C03640=1043.062,430.880,361.254,175.358,44.997,159.099
C03641=1043.073,431.124,361.204,175.371,45.006,159.102
C03642=1043.084,431.369,361.154,175.384,45.014,159.106
C03643=1043.096,431.614,361.104,175.397,45.023,159.110
C03644=1043.107,431.859,361.054,175.411,45.031,159.113
C03645=1043.119,432.104,361.004,175.424,45.040,159.117
C03646=1043.130,432.348,360.954,175.437,45.048,159.121
C03647=1043.142,432.593,360.904,175.450,45.057,159.125
C03648=1043.153,432.837,360.853,175.463,45.065,159.128
C03649=1043.165,433.082,360.803,175.477,45.074,159.132
C03650=1043.177,433.326,360.752,175.491,45.083,159.136
C03651=1043.188,433.571,360.701,175.504,45.092,159.140
C03652=1043.200,433.815,360.652,175.517,45.100,159.144
C03653=1043.212,434.060,360.601,175.531,45.109,159.147
C03654=1043.223,434.288,360.554,175.543,45.117,159.151
C03655=1043.234,434.517,360.506,175.556,45.125,159.155
C03656=1043.245,434.745,360.459,175.570,45.133,159.158
C03657=1043.256,434.972,360.411,175.581,45.142,159.162
C03658=1043.267,435.201,360.364,175.595,45.150,159.166
C03659=1043.278,435.429,360.317,175.608,45.158,159.169
C03660=1043.290,435.657,360.269,175.621,45.166,159.173
C03661=1043.301,435.885,360.222,175.634,45.175,159.177
C03662=1043.312,436.130,360.171,175.647,45.184,159.181
C03663=1043.324,436.374,360.119,175.662,45.193,159.185
C03664=1043.335,436.618,360.068,175.675,45.202,159.189
C03665=1043.348,436.862,360.018,175.690,45.211,159.193
C03666=1043.360,437.107,359.966,175.704,45.220,159.197
C03667=1043.372,437.351,359.915,175.718,45.229,159.201
C03668=1043.384,437.597,359.863,175.732,45.238,159.205
C03669=1043.397,437.840,359.811,175.747,45.247,159.209
C03670=1043.408,438.085,359.759,175.761,45.257,159.213
C03671=1043.420,438.329,359.708,175.775,45.266,159.217
C03672=1043.432,438.573,359.656,175.790,45.275,159.222
C03673=1043.445,438.818,359.605,175.805,45.284,159.226
C03674=1043.457,439.061,359.553,175.820,45.294,159.230
C03675=1043.469,439.306,359.502,175.835,45.303,159.234
C03676=1043.481,439.550,359.449,175.848,45.313,159.238
C03677=1043.494,439.794,359.397,175.863,45.322,159.243
C03678=1043.506,440.039,359.346,175.878,45.332,159.247
C03679=1043.518,440.283,359.293,175.893,45.341,159.251
C03680=1043.531,440.527,359.241,175.908,45.350,159.256
C03681=1043.543,440.771,359.189,175.923,45.360,159.260
C03682=1043.555,441.015,359.137,175.938,45.370,159.264
C03683=1043.568,441.260,359.084,175.953,45.379,159.269
C03684=1043.580,441.504,359.032,175.969,45.389,159.273
C03685=1043.593,441.748,358.980,175.984,45.399,159.277
C03686=1043.605,441.992,358.928,176.000,45.408,159.282
C03687=1043.618,442.236,358.874,176.015,45.418,159.286
C03688=1043.631,442.480,358.822,176.030,45.428,159.291
C03689=1043.643,442.725,358.770,176.045,45.437,159.295
C03690=1043.655,442.968,358.716,176.062,45.447,159.300
C03691=1043.668,443.213,358.664,176.077,45.457,159.304
C03692=1043.681,443.457,358.611,176.092,45.467,159.309
C03693=1043.694,443.700,358.558,176.109,45.476,159.313
C03694=1043.706,443.945,358.505,176.124,45.486,159.318
C03695=1043.719,444.189,358.452,176.140,45.496,159.322
C03696=1043.732,444.433,358.399,176.156,45.506,159.327
C03697=1043.746,444.677,358.346,176.171,45.516,159.332
C03698=1043.758,444.920,358.293,176.188,45.527,159.337
C03699=1043.772,445.162,358.240,176.205,45.536,159.341
C03700=1043.784,445.405,358.187,176.220,45.546,159.346
C03701=1043.799,445.650,358.135,176.237,45.556,159.350
C03702=1043.813,445.893,358.084,176.253,45.566,159.355
C03703=1043.828,446.136,358.032,176.269,45.575,159.360
C03704=1043.845,446.380,357.982,176.286,45.585,159.364
C03705=1043.861,446.624,357.931,176.302,45.594,159.369
C03706=1043.879,446.867,357.882,176.319,45.603,159.373
C03707=1043.896,447.112,357.833,176.336,45.613,159.378
C03708=1043.915,447.355,357.784,176.353,45.621,159.382
C03709=1043.934,447.601,357.735,176.369,45.630,159.387
C03710=1043.954,447.845,357.687,176.386,45.639,159.391
C03711=1043.974,448.089,357.641,176.403,45.648,159.396
C03712=1043.995,448.334,357.593,176.420,45.656,159.400
C03713=1044.016,448.578,357.547,176.438,45.665,159.404
C03714=1044.054,448.991,357.470,176.467,45.678,159.412
C03715=1044.094,449.404,357.395,176.496,45.692,159.419
C03716=1044.135,449.817,357.321,176.526,45.706,159.426
C03717=1044.178,450.231,357.248,176.556,45.718,159.433
C03718=1044.204,450.476,357.205,176.574,45.726,159.438
C03719=1044.231,450.722,357.163,176.591,45.733,159.442
C03720=1044.259,450.968,357.122,176.610,45.741,159.446
C03721=1044.287,451.213,357.081,176.627,45.748,159.450
C03722=1043.984,451.252,356.769,176.629,45.829,159.475
C03723=1043.956,451.007,356.810,176.612,45.822,159.470
C03724=1043.927,450.761,356.851,176.593,45.815,159.466
C03725=1043.901,450.516,356.893,176.575,45.808,159.462
C03726=1043.874,450.271,356.936,176.558,45.800,159.458
C03727=1043.833,449.874,357.005,176.528,45.788,159.451
C03728=1043.793,449.476,357.076,176.500,45.775,159.444
C03729=1043.754,449.080,357.149,176.471,45.763,159.437
C03730=1043.717,448.682,357.223,176.443,45.749,159.430
C03731=1043.695,448.438,357.268,176.426,45.741,159.426
C03732=1043.674,448.193,357.315,176.408,45.733,159.421
C03733=1043.654,447.949,357.362,176.391,45.724,159.417
C03734=1043.633,447.704,357.410,176.374,45.716,159.412
C03735=1043.614,447.460,357.458,176.358,45.706,159.408
C03736=1043.595,447.216,357.506,176.341,45.698,159.403
C03737=1043.577,446.972,357.554,176.324,45.689,159.399
C03738=1043.559,446.727,357.605,176.307,45.680,159.394
C03739=1043.542,446.484,357.654,176.290,45.671,159.390
C03740=1043.526,446.240,357.705,176.274,45.662,159.385
C03741=1043.511,445.997,357.756,176.257,45.652,159.381
C03742=1043.496,445.753,357.807,176.241,45.643,159.376
C03743=1043.481,445.510,357.859,176.225,45.633,159.372
C03744=1043.467,445.266,357.912,176.208,45.623,159.367
C03745=1043.454,445.023,357.964,176.193,45.613,159.362
C03746=1043.441,444.781,358.017,176.176,45.603,159.358
C03747=1043.421,444.396,358.101,176.151,45.587,159.350
C03748=1043.400,444.010,358.184,176.125,45.572,159.343
C03749=1043.380,443.625,358.269,176.100,45.556,159.336
C03750=1043.360,443.240,358.352,176.075,45.541,159.329
C03751=1043.347,442.995,358.405,176.060,45.531,159.324
C03752=1043.334,442.752,358.457,176.044,45.522,159.320
C03753=1043.322,442.508,358.510,176.028,45.512,159.315
C03754=1043.309,442.264,358.563,176.013,45.502,159.310
C03755=1043.296,442.020,358.615,175.998,45.493,159.306
C03756=1043.284,441.776,358.667,175.982,45.483,159.302
C03757=1043.271,441.532,358.721,175.967,45.474,159.297
C03758=1043.259,441.288,358.773,175.952,45.464,159.293
C03759=1043.246,441.043,358.825,175.936,45.454,159.288
C03760=1043.234,440.800,358.877,175.921,45.445,159.284
C03761=1043.221,440.555,358.930,175.906,45.436,159.280
C03762=1043.209,440.311,358.982,175.891,45.426,159.275
C03763=1043.197,440.067,359.033,175.876,45.417,159.271
C03764=1043.184,439.822,359.086,175.861,45.407,159.267
C03765=1043.172,439.578,359.138,175.846,45.398,159.263
C03766=1043.160,439.334,359.190,175.832,45.389,159.258
C03767=1043.147,439.089,359.242,175.817,45.379,159.254
C03768=1043.135,438.845,359.294,175.802,45.370,159.250
C03769=1043.123,438.601,359.345,175.788,45.361,159.246
C03770=1043.111,438.357,359.397,175.773,45.351,159.241
C03771=1043.099,438.112,359.449,175.758,45.342,159.237
C03772=1043.087,437.868,359.500,175.744,45.334,159.233
C03773=1043.074,437.624,359.552,175.730,45.324,159.229
C03774=1043.062,437.380,359.603,175.715,45.315,159.225
C03775=1043.051,437.135,359.655,175.701,45.306,159.221
C03776=1043.039,436.891,359.706,175.687,45.297,159.217
C03777=1043.027,436.646,359.757,175.672,45.288,159.213
C03778=1043.014,436.402,359.808,175.659,45.279,159.209
C03779=1043.002,436.157,359.860,175.644,45.270,159.205
C03780=1042.990,435.913,359.911,175.631,45.261,159.201
C03781=1042.979,435.668,359.962,175.616,45.252,159.197
C03782=1042.967,435.423,360.013,175.603,45.243,159.193
C03783=1042.951,435.108,360.079,175.584,45.232,159.188
C03784=1042.936,434.791,360.145,175.567,45.221,159.183
C03785=1042.920,434.475,360.210,175.548,45.209,159.178
C03786=1042.905,434.158,360.276,175.531,45.198,159.173
C03787=1042.894,433.913,360.326,175.517,45.189,159.169
C03788=1042.881,433.669,360.377,175.504,45.181,159.165
C03789=1042.870,433.424,360.428,175.490,45.172,159.161
C03790=1042.858,433.180,360.477,175.476,45.164,159.157
C03791=1042.847,432.935,360.528,175.463,45.155,159.153
C03792=1042.835,432.691,360.578,175.450,45.147,159.150
C03793=1042.823,432.446,360.628,175.437,45.138,159.146
C03794=1042.812,432.201,360.679,175.424,45.130,159.142
C03795=1042.800,431.956,360.729,175.411,45.121,159.138
C03796=1042.789,431.712,360.779,175.396,45.113,159.135
C03797=1042.777,431.467,360.829,175.383,45.104,159.131
C03798=1042.766,431.223,360.880,175.370,45.096,159.127
C03799=1042.754,430.978,360.930,175.357,45.087,159.124
C03800=1042.743,430.733,360.979,175.345,45.079,159.120
C03801=1042.732,430.488,361.030,175.332,45.071,159.116
C03802=1042.720,430.244,361.079,175.319,45.062,159.113
C03803=1042.709,429.998,361.129,175.306,45.054,159.109
C03804=1042.697,429.754,361.179,175.293,45.046,159.105
C03805=1042.686,429.509,361.229,175.280,45.037,159.102
C03806=1042.675,429.265,361.279,175.267,45.029,159.098
C03807=1042.664,429.020,361.328,175.255,45.021,159.095
C03808=1042.653,428.774,361.378,175.243,45.013,159.091
C03809=1042.641,428.530,361.427,175.229,45.005,159.087
C03810=1042.630,428.285,361.477,175.217,44.997,159.084
C03811=1042.619,428.040,361.526,175.205,44.989,159.081
C03812=1042.608,427.796,361.575,175.192,44.981,159.077
C03813=1042.597,427.551,361.625,175.179,44.973,159.074
C03814=1042.586,427.306,361.674,175.168,44.964,159.070
C03815=1042.574,427.061,361.723,175.155,44.957,159.067
C03816=1042.563,426.816,361.771,175.142,44.949,159.063
C03817=1042.552,426.571,361.821,175.131,44.941,159.060
C03818=1042.541,426.326,361.870,175.118,44.933,159.056
C03819=1042.530,426.081,361.919,175.106,44.925,159.053
C03820=1042.519,425.836,361.968,175.094,44.917,159.050
C03821=1042.508,425.591,362.017,175.082,44.909,159.046
C03822=1042.497,425.347,362.065,175.070,44.902,159.043
C03823=1042.487,425.101,362.114,175.058,44.894,159.040
C03824=1042.475,424.856,362.163,175.045,44.886,159.036
C03825=1042.464,424.611,362.212,175.034,44.878,159.033
C03826=1042.454,424.366,362.260,175.022,44.870,159.030
C03827=1042.443,424.121,362.309,175.010,44.863,159.026
C03828=1042.432,423.876,362.358,174.998,44.855,159.023
C03829=1042.421,423.631,362.406,174.987,44.847,159.020
C03830=1042.410,423.386,362.454,174.974,44.840,159.017
C03831=1042.399,423.141,362.502,174.963,44.833,159.013
C03832=1042.388,422.895,362.550,174.952,44.825,159.010
C03833=1042.377,422.651,362.599,174.941,44.817,159.007
C03834=1042.366,422.405,362.647,174.928,44.810,159.004
C03835=1042.356,422.161,362.694,174.917,44.803,159.001
C03836=1042.345,421.915,362.743,174.905,44.795,158.997
C03837=1042.334,421.671,362.791,174.894,44.787,158.994
C03838=1042.323,421.425,362.839,174.883,44.780,158.991
C03839=1042.314,421.205,362.882,174.872,44.773,158.988
C03840=1042.304,420.985,362.925,174.862,44.767,158.986
C03841=1042.295,420.765,362.968,174.852,44.760,158.983
C03842=1042.286,420.546,363.011,174.842,44.754,158.980
C03843=1042.276,420.327,363.054,174.832,44.747,158.977
C03844=1042.267,420.106,363.097,174.822,44.740,158.974
C03845=1042.257,419.886,363.140,174.811,44.734,158.972
C03846=1042.248,419.666,363.182,174.802,44.728,158.969
C03847=1042.237,419.421,363.230,174.791,44.720,158.966
C03848=1042.227,419.176,363.278,174.779,44.713,158.963
C03849=1042.217,418.930,363.325,174.768,44.705,158.960
C03850=1042.206,418.686,363.373,174.757,44.699,158.957
C03851=1042.196,418.440,363.420,174.747,44.691,158.954
C03852=1042.186,418.195,363.467,174.736,44.684,158.951
C03853=1042.175,417.950,363.515,174.725,44.677,158.948
C03854=1042.165,417.704,363.562,174.714,44.670,158.945
C03855=1042.154,417.459,363.609,174.703,44.663,158.942
C03856=1042.144,417.213,363.656,174.692,44.656,158.939
C03857=1042.133,416.968,363.703,174.681,44.649,158.936
C03858=1042.123,416.723,363.751,174.671,44.642,158.933
C03859=1042.112,416.478,363.797,174.660,44.635,158.930
C03860=1042.102,416.233,363.844,174.649,44.628,158.927
C03861=1042.092,415.987,363.892,174.638,44.621,158.924
C03862=1042.081,415.741,363.938,174.628,44.614,158.922
C03863=1042.071,415.496,363.985,174.618,44.607,158.919
C03864=1042.061,415.251,364.032,174.607,44.601,158.916
C03865=1042.051,415.005,364.078,174.597,44.594,158.913
C03866=1042.041,414.760,364.126,174.586,44.587,158.910
C03867=1042.030,414.514,364.172,174.575,44.580,158.907
C03868=1042.020,414.269,364.219,174.565,44.573,158.905
C03869=1042.010,414.023,364.265,174.555,44.566,158.902
C03870=1042.000,413.778,364.312,174.545,44.559,158.899
C03871=1041.989,413.532,364.358,174.534,44.553,158.896
C03872=1041.980,413.288,364.405,174.525,44.546,158.893
C03873=1041.970,413.042,364.452,174.514,44.540,158.891
C03874=1041.960,412.796,364.498,174.504,44.532,158.888
C03875=1041.949,412.550,364.544,174.494,44.526,158.885
C03876=1041.940,412.306,364.591,174.484,44.520,158.883
C03877=1041.930,412.060,364.637,174.473,44.513,158.880
C03878=1041.919,411.814,364.683,174.463,44.506,158.877
C03879=1041.910,411.569,364.730,174.453,44.500,158.874
C03880=1041.899,411.323,364.775,174.443,44.493,158.872
C03881=1041.889,411.078,364.822,174.434,44.487,158.869
C03882=1041.880,410.832,364.867,174.423,44.480,158.866
C03883=1041.869,410.586,364.913,174.414,44.474,158.864
C03884=1041.859,410.341,364.959,174.403,44.467,158.861
C03885=1041.849,410.096,365.005,174.393,44.461,158.858
C03886=1041.840,409.849,365.050,174.384,44.455,158.856
C03887=1041.830,409.604,365.096,174.374,44.448,158.853
C03888=1041.820,409.358,365.143,174.364,44.442,158.851
C03889=1041.810,409.113,365.187,174.355,44.436,158.848
C03890=1041.799,408.867,365.233,174.345,44.429,158.845
C03891=1041.790,408.621,365.279,174.335,44.423,158.843
C03892=1041.780,408.376,365.325,174.325,44.416,158.840
C03893=1041.771,408.130,365.370,174.316,44.410,158.838
C03894=1041.761,407.885,365.416,174.306,44.404,158.835
C03895=1041.750,407.639,365.461,174.297,44.398,158.833
C03896=1041.741,407.394,365.507,174.287,44.391,158.830
C03897=1041.731,407.148,365.552,174.277,44.385,158.828
C03898=1041.721,406.902,365.597,174.268,44.379,158.825
C03899=1041.713,406.686,365.637,174.260,44.373,158.823
C03900=1041.704,406.471,365.677,174.251,44.368,158.821
C03901=1041.696,406.255,365.716,174.243,44.363,158.819
C03902=1041.688,406.039,365.757,174.235,44.357,158.816
C03903=1041.679,405.823,365.796,174.226,44.352,158.814
C03904=1041.671,405.607,365.836,174.218,44.346,158.812
C03905=1041.662,405.392,365.875,174.211,44.341,158.810
C03906=1041.655,405.176,365.915,174.202,44.335,158.808
C03907=1041.645,404.930,365.960,174.192,44.330,158.805
C03908=1041.635,404.685,366.005,174.183,44.324,158.803
C03909=1041.626,404.439,366.050,174.175,44.318,158.800
C03910=1041.616,404.194,366.095,174.166,44.312,158.798
C03911=1041.606,403.947,366.140,174.156,44.305,158.796
C03912=1041.597,403.701,366.185,174.147,44.299,158.793
C03913=1041.588,403.455,366.230,174.138,44.294,158.791
C03914=1041.578,403.210,366.274,174.129,44.288,158.788
C03915=1041.568,402.964,366.319,174.120,44.282,158.786
C03916=1041.559,402.718,366.363,174.111,44.276,158.784
C03917=1041.550,402.472,366.409,174.101,44.270,158.781
C03918=1041.541,402.227,366.453,174.092,44.264,158.779
C03919=1041.531,401.981,366.497,174.083,44.259,158.777
C03920=1041.522,401.735,366.541,174.074,44.253,158.774
C03921=1041.512,401.490,366.586,174.066,44.247,158.772
C03922=1041.503,401.244,366.630,174.057,44.241,158.770
C03923=1041.493,400.998,366.675,174.048,44.235,158.767
C03924=1041.484,400.752,366.719,174.039,44.230,158.765
C03925=1041.474,400.506,366.763,174.030,44.224,158.763
C03926=1041.465,400.260,366.807,174.022,44.218,158.760
C03927=1041.456,400.015,366.852,174.013,44.213,158.758
C03928=1041.446,399.769,366.896,174.004,44.207,158.756
C03929=1041.437,399.523,366.940,173.995,44.201,158.754
C03930=1041.428,399.277,366.984,173.987,44.196,158.751
C03931=1041.419,399.031,367.028,173.978,44.190,158.749
C03932=1041.409,398.785,367.072,173.969,44.184,158.747
C03933=1041.400,398.539,367.116,173.960,44.179,158.745
C03934=1041.391,398.293,367.160,173.952,44.173,158.742
C03935=1041.382,398.047,367.204,173.943,44.167,158.740
C03936=1041.373,397.802,367.248,173.934,44.162,158.738
C03937=1041.363,397.556,367.292,173.926,44.156,158.736
C03938=1041.353,397.310,367.335,173.917,44.151,158.734
C03939=1041.345,397.064,367.379,173.909,44.146,158.732
C03940=1041.335,396.818,367.423,173.901,44.140,158.729
C03941=1041.327,396.572,367.466,173.892,44.135,158.727
C03942=1041.317,396.326,367.510,173.884,44.129,158.725
C03943=1041.309,396.080,367.553,173.875,44.124,158.723
C03944=1041.299,395.834,367.598,173.866,44.118,158.721
C03945=1041.290,395.589,367.641,173.859,44.113,158.719
C03946=1041.281,395.343,367.684,173.850,44.108,158.716
C03947=1041.272,395.097,367.728,173.842,44.102,158.714
C03948=1041.263,394.851,367.771,173.833,44.097,158.712
C03949=1041.253,394.605,367.814,173.825,44.091,158.710
C03950=1041.245,394.359,367.857,173.817,44.086,158.708
C03951=1041.236,394.112,367.901,173.809,44.081,158.706
C03952=1041.227,393.867,367.945,173.800,44.076,158.704
C03953=1041.218,393.621,367.987,173.792,44.071,158.702
C03954=1041.208,393.374,368.030,173.784,44.066,158.700
C03955=1041.200,393.129,368.074,173.776,44.060,158.698
C03956=1041.190,392.883,368.117,173.767,44.055,158.696
C03957=1041.182,392.637,368.160,173.760,44.050,158.694
C03958=1041.173,392.390,368.203,173.752,44.045,158.692
C03959=1041.158,391.979,368.275,173.739,44.036,158.688
C03960=1041.142,391.566,368.346,173.725,44.027,158.685
C03961=1041.128,391.155,368.419,173.712,44.018,158.681
C03962=1041.113,390.742,368.490,173.698,44.010,158.678
C03963=1041.104,390.497,368.533,173.690,44.005,158.676
C03964=1041.096,390.250,368.575,173.682,44.000,158.674
C03965=1041.086,390.004,368.618,173.674,43.995,158.672
C03966=1041.078,389.758,368.661,173.666,43.990,158.670
C03967=1041.069,389.512,368.703,173.658,43.985,158.668
C03968=1041.060,389.266,368.746,173.651,43.980,158.666
C03969=1041.051,389.020,368.788,173.642,43.975,158.664
C03970=1041.043,388.774,368.831,173.635,43.970,158.662
C03971=1041.033,388.527,368.873,173.627,43.966,158.661
C03972=1041.025,388.281,368.916,173.620,43.960,158.658
C03973=1041.015,388.035,368.958,173.611,43.956,158.657
C03974=1041.007,387.788,369.001,173.604,43.951,158.655
C03975=1040.998,387.542,369.042,173.596,43.946,158.653
C03976=1040.989,387.296,369.085,173.589,43.941,158.651
C03977=1040.980,387.050,369.126,173.580,43.936,158.649
C03978=1040.972,386.804,369.169,173.573,43.931,158.647
C03979=1040.963,386.557,369.211,173.565,43.927,158.645
C03980=1040.954,386.311,369.253,173.558,43.922,158.643
C03981=1040.945,386.065,369.294,173.551,43.917,158.642
C03982=1040.937,385.819,369.337,173.543,43.912,158.640
C03983=1040.928,385.573,369.379,173.535,43.908,158.638
C03984=1040.919,385.327,369.421,173.527,43.903,158.636
C03985=1040.910,385.080,369.462,173.520,43.898,158.634
C03986=1040.901,384.834,369.504,173.512,43.893,158.632
C03987=1040.893,384.587,369.546,173.505,43.889,158.630
C03988=1040.885,384.342,369.588,173.498,43.884,158.629
C03989=1040.876,384.095,369.630,173.490,43.880,158.627
C03990=1040.867,383.849,369.671,173.483,43.875,158.625
C03991=1040.859,383.602,369.714,173.476,43.870,158.623
C03992=1040.850,383.356,369.755,173.467,43.865,158.621
C03993=1040.841,383.110,369.797,173.460,43.861,158.620
C03994=1040.832,382.864,369.838,173.453,43.856,158.618
C03995=1040.824,382.617,369.881,173.445,43.852,158.616
C03996=1040.816,382.371,369.922,173.438,43.847,158.614
C03997=1040.807,382.124,369.963,173.431,43.843,158.612
C03998=1040.798,381.878,370.005,173.423,43.838,158.611
C03999=1040.790,381.632,370.046,173.416,43.834,158.609
C04000=1040.782,381.386,370.088,173.409,43.829,158.607
C04001=1040.773,381.139,370.129,173.402,43.825,158.605
C04002=1040.765,380.893,370.171,173.394,43.820,158.604
C04003=1040.756,380.646,370.212,173.387,43.816,158.602
C04004=1040.748,380.400,370.253,173.381,43.811,158.600
C04005=1040.740,380.154,370.295,173.374,43.806,158.598
C04006=1040.732,379.907,370.336,173.366,43.802,158.597
C04007=1040.723,379.661,370.378,173.359,43.798,158.595
C04008=1040.715,379.415,370.418,173.352,43.793,158.593
C04009=1040.706,379.168,370.460,173.345,43.789,158.592
C04010=1040.698,378.922,370.501,173.338,43.784,158.590
C04011=1040.690,378.675,370.542,173.330,43.780,158.588
C04012=1040.681,378.430,370.583,173.323,43.775,158.586
C04013=1040.672,378.183,370.624,173.316,43.771,158.585
C04014=1040.664,377.936,370.665,173.310,43.767,158.583
C04015=1040.651,377.558,370.728,173.299,43.761,158.581
C04016=1040.638,377.180,370.790,173.288,43.754,158.578
C04017=1040.625,376.802,370.853,173.277,43.747,158.576
C04018=1040.612,376.424,370.915,173.267,43.741,158.573
C04019=1040.604,376.177,370.956,173.260,43.737,158.572
C04020=1040.596,375.931,370.997,173.253,43.733,158.570
C04021=1040.588,375.685,371.037,173.245,43.728,158.568
C04022=1040.579,375.438,371.078,173.239,43.724,158.567
C04023=1040.570,375.192,371.118,173.232,43.720,158.565
C04024=1040.562,374.945,371.159,173.225,43.716,158.563
C04025=1040.554,374.698,371.200,173.218,43.712,158.562
C04026=1040.546,374.452,371.240,173.212,43.707,158.560
C04027=1040.538,374.205,371.280,173.205,43.703,158.559
C04028=1040.530,373.959,371.321,173.198,43.699,158.557
C04029=1040.520,373.712,371.361,173.191,43.695,158.555
C04030=1040.512,373.466,371.402,173.185,43.691,158.554
C04031=1040.505,373.219,371.442,173.178,43.687,158.552
C04032=1040.497,372.973,371.483,173.171,43.683,158.551
C04033=1040.489,372.726,371.523,173.165,43.679,158.549
C04034=1040.481,372.479,371.563,173.158,43.674,158.547
C04035=1040.472,372.233,371.604,173.151,43.671,158.546
C04036=1040.464,371.987,371.644,173.145,43.667,158.545
C04037=1040.456,371.740,371.684,173.138,43.662,158.543
C04038=1040.448,371.493,371.725,173.131,43.659,158.541
C04039=1040.440,371.246,371.765,173.125,43.654,158.540
C04040=1040.431,371.000,371.805,173.118,43.650,158.538
C04041=1040.424,370.754,371.845,173.112,43.647,158.537
C04042=1040.416,370.507,371.885,173.105,43.642,158.535
C04043=1040.408,370.260,371.925,173.098,43.638,158.534
C04044=1040.399,370.014,371.965,173.092,43.635,158.532
C04045=1040.391,369.766,372.005,173.085,43.631,158.531
C04046=1040.382,369.520,372.045,173.078,43.627,158.529
C04047=1040.375,369.273,372.085,173.072,43.623,158.528
C04048=1040.366,369.027,372.124,173.065,43.619,158.526
C04049=1040.358,368.780,372.164,173.060,43.615,158.525
C04050=1040.350,368.533,372.203,173.053,43.611,158.523
C04051=1040.342,368.286,372.243,173.047,43.607,158.522
C04052=1040.334,368.040,372.283,173.040,43.604,158.520
C04053=1040.326,367.793,372.322,173.033,43.600,158.519
C04054=1040.318,367.546,372.362,173.027,43.596,158.517
C04055=1040.310,367.299,372.402,173.020,43.592,158.516
C04056=1040.301,367.053,372.441,173.014,43.588,158.514
C04057=1040.294,366.806,372.481,173.008,43.585,158.513
C04058=1040.286,366.560,372.520,173.002,43.581,158.512
C04059=1040.277,366.313,372.559,172.995,43.577,158.510
C04060=1040.270,366.066,372.599,172.989,43.574,158.509
C04061=1040.261,365.820,372.638,172.982,43.570,158.507
C04062=1040.253,365.573,372.678,172.976,43.566,158.506
C04063=1040.245,365.326,372.718,172.970,43.562,158.504
C04064=1040.238,365.079,372.757,172.964,43.559,158.503
C04065=1040.230,364.833,372.796,172.958,43.555,158.502
C04066=1040.222,364.586,372.836,172.951,43.551,158.500
C04067=1040.214,364.339,372.875,172.946,43.548,158.499
C04068=1040.206,364.092,372.914,172.939,43.544,158.497
C04069=1040.198,363.846,372.953,172.933,43.540,158.496
C04070=1040.191,363.599,372.993,172.926,43.537,158.495
C04071=1040.179,363.240,373.050,172.918,43.532,158.493
C04072=1040.167,362.883,373.106,172.909,43.526,158.491
C04073=1040.157,362.525,373.163,172.900,43.521,158.489
C04074=1040.145,362.167,373.219,172.891,43.516,158.487
C04075=1040.137,361.920,373.259,172.885,43.512,158.485
C04076=1040.129,361.673,373.298,172.879,43.509,158.484
C04077=1040.121,361.426,373.337,172.873,43.505,158.482
C04078=1040.113,361.179,373.375,172.867,43.501,158.481
C04079=1040.105,360.933,373.414,172.860,43.498,158.480
C04080=1040.098,360.686,373.454,172.855,43.494,158.478
C04081=1040.089,360.439,373.492,172.849,43.491,158.477
C04082=1040.082,360.192,373.531,172.842,43.488,158.476
C04083=1040.074,359.945,373.569,172.837,43.484,158.474
C04084=1040.066,359.698,373.607,172.831,43.480,158.473
C04085=1040.058,359.452,373.647,172.824,43.477,158.472
C04086=1040.050,359.204,373.686,172.819,43.474,158.470
C04087=1040.043,358.958,373.724,172.813,43.470,158.469
C04088=1040.035,358.711,373.763,172.806,43.467,158.468
C04089=1040.027,358.464,373.801,172.801,43.464,158.467
C04090=1040.019,358.217,373.840,172.795,43.460,158.465
C04091=1040.011,357.970,373.878,172.789,43.456,158.464
C04092=1040.003,357.723,373.916,172.783,43.453,158.463
C04093=1039.996,357.477,373.955,172.777,43.450,158.461
C04094=1039.988,357.229,373.994,172.772,43.446,158.460
C04095=1039.981,356.983,374.032,172.766,43.443,158.459
C04096=1039.973,356.735,374.071,172.759,43.440,158.457
C04097=1039.965,356.489,374.109,172.754,43.436,158.456
C04098=1039.958,356.242,374.147,172.748,43.433,158.455
C04099=1039.950,355.994,374.185,172.742,43.430,158.454
C04100=1039.942,355.748,374.223,172.736,43.426,158.452
C04101=1039.934,355.501,374.262,172.730,43.424,158.451
C04102=1039.927,355.254,374.299,172.725,43.420,158.450
C04103=1039.918,355.007,374.338,172.719,43.417,158.449
C04104=1039.910,354.760,374.376,172.714,43.413,158.447
C04105=1039.903,354.513,374.413,172.707,43.410,158.446
C04106=1039.895,354.266,374.452,172.702,43.407,158.445
C04107=1039.887,354.019,374.490,172.696,43.404,158.444
C04108=1039.880,353.772,374.528,172.690,43.401,158.443
C04109=1039.872,353.525,374.566,172.685,43.397,158.441
C04110=1039.865,353.278,374.604,172.679,43.394,158.440
C04111=1039.857,353.031,374.642,172.673,43.391,158.439
C04112=1039.849,352.783,374.680,172.667,43.388,158.438
C04113=1039.841,352.537,374.718,172.662,43.385,158.436
C04114=1039.834,352.290,374.755,172.656,43.382,158.435
C04115=1039.826,352.043,374.794,172.651,43.378,158.434
C04116=1039.818,351.796,374.831,172.645,43.375,158.433
C04117=1039.811,351.549,374.869,172.640,43.372,158.432
C04118=1039.804,351.302,374.907,172.634,43.369,158.430
C04119=1039.796,351.055,374.945,172.629,43.366,158.429
C04120=1039.788,350.808,374.983,172.623,43.362,158.428
C04121=1039.780,350.561,375.020,172.617,43.360,158.427
C04122=1039.773,350.314,375.058,172.611,43.356,158.426
C04123=1039.766,350.067,375.095,172.606,43.353,158.424
C04124=1039.758,349.820,375.133,172.600,43.351,158.423
C04125=1039.751,349.573,375.171,172.595,43.347,158.422
C04126=1039.742,349.325,375.208,172.589,43.344,158.421
C04127=1039.732,348.974,375.262,172.581,43.340,158.419
C04128=1039.721,348.621,375.315,172.574,43.336,158.418
C04129=1039.711,348.270,375.368,172.566,43.331,158.416
C04130=1039.700,347.917,375.421,172.558,43.327,158.414
C04131=1039.692,347.670,375.458,172.553,43.324,158.413
C04132=1039.684,347.423,375.496,172.547,43.321,158.412
C04133=1039.677,347.176,375.533,172.542,43.318,158.411
C04134=1039.669,346.929,375.570,172.537,43.315,158.410
C04135=1039.662,346.682,375.608,172.531,43.312,158.409
C04136=1039.655,346.435,375.645,172.526,43.309,158.408
C04137=1039.647,346.188,375.682,172.520,43.306,158.406
C04138=1039.639,345.940,375.720,172.515,43.303,158.405
C04139=1039.631,345.693,375.756,172.510,43.301,158.404
C04140=1039.625,345.447,375.794,172.504,43.298,158.403
C04141=1039.617,345.199,375.831,172.499,43.295,158.402
C04142=1039.609,344.953,375.868,172.493,43.292,158.401
C04143=1039.602,344.705,375.905,172.488,43.289,158.400
C04144=1039.594,344.458,375.942,172.483,43.286,158.399
C04145=1039.587,344.211,375.979,172.478,43.283,158.398
C04146=1039.580,343.963,376.016,172.473,43.280,158.397
C04147=1039.572,343.716,376.053,172.468,43.278,158.395
C04148=1039.564,343.469,376.090,172.462,43.275,158.394
C04149=1039.557,343.222,376.127,172.457,43.272,158.393
C04150=1039.549,342.975,376.164,172.452,43.269,158.392
C04151=1039.542,342.727,376.201,172.446,43.266,158.391
C04152=1039.535,342.480,376.238,172.441,43.263,158.390
C04153=1039.528,342.233,376.274,172.435,43.261,158.389
C04154=1039.520,341.986,376.311,172.430,43.258,158.388
C04155=1039.513,341.759,376.345,172.426,43.255,158.387
C04156=1039.507,341.531,376.379,172.421,43.252,158.386
C04157=1039.500,341.304,376.413,172.417,43.250,158.385
C04158=1039.493,341.076,376.446,172.411,43.248,158.384
C04159=1039.486,340.849,376.480,172.407,43.245,158.383
C04160=1039.479,340.622,376.513,172.402,43.242,158.382
C04161=1039.473,340.395,376.547,172.397,43.240,158.381
C04162=1039.465,340.167,376.580,172.393,43.238,158.380
C04163=1039.459,339.920,376.617,172.387,43.235,158.379
C04164=1039.451,339.673,376.654,172.382,43.232,158.378
C04165=1039.443,339.426,376.690,172.377,43.230,158.377
C04166=1039.435,339.178,376.726,172.372,43.227,158.376
C04167=1039.428,338.930,376.763,172.367,43.224,158.375
C04168=1039.421,338.684,376.799,172.362,43.222,158.374
C04169=1039.413,338.437,376.836,172.357,43.219,158.373
C04170=1039.406,338.189,376.873,172.351,43.216,158.372
C04171=1039.399,337.942,376.909,172.347,43.213,158.371
C04172=1039.392,337.695,376.945,172.342,43.211,158.370
C04173=1039.384,337.447,376.981,172.337,43.208,158.369
C04174=1039.377,337.200,377.018,172.331,43.205,158.368
C04175=1039.370,336.953,377.054,172.326,43.203,158.367
C04176=1039.362,336.705,377.090,172.322,43.200,158.366
C04177=1039.355,336.458,377.126,172.317,43.198,158.365
C04178=1039.347,336.211,377.162,172.311,43.195,158.364
C04179=1039.341,335.963,377.199,172.306,43.193,158.363
C04180=1039.333,335.717,377.234,172.302,43.190,158.362
C04181=1039.326,335.469,377.271,172.297,43.187,158.361
C04182=1039.318,335.222,377.307,172.291,43.184,158.360
C04183=1039.307,334.826,377.364,172.284,43.181,158.358
C04184=1039.295,334.431,377.422,172.276,43.176,158.357
C04185=1039.283,334.036,377.479,172.268,43.173,158.355
C04186=1039.272,333.640,377.537,172.260,43.168,158.354
C04187=1039.265,333.393,377.573,172.255,43.166,158.353
C04188=1039.257,333.146,377.609,172.251,43.164,158.352
C04189=1039.250,332.898,377.644,172.245,43.161,158.351
C04190=1039.243,332.651,377.680,172.240,43.159,158.350
C04191=1039.236,332.403,377.715,172.236,43.156,158.349
C04192=1039.228,332.156,377.752,172.231,43.154,158.348
C04193=1039.221,331.909,377.787,172.225,43.151,158.347
C04194=1039.214,331.661,377.823,172.221,43.148,158.346
C04195=1039.206,331.415,377.858,172.216,43.146,158.345
C04196=1039.199,331.167,377.894,172.211,43.144,158.344
C04197=1039.191,330.920,377.929,172.207,43.141,158.343
C04198=1039.184,330.672,377.965,172.202,43.139,158.342
C04199=1039.177,330.425,378.001,172.197,43.137,158.341
C04200=1039.170,330.178,378.036,172.192,43.134,158.340
C04201=1039.163,329.930,378.072,172.187,43.131,158.339
C04202=1039.156,329.683,378.107,172.182,43.129,158.338
C04203=1039.148,329.436,378.144,172.178,43.127,158.338
C04204=1039.141,329.188,378.179,172.173,43.124,158.337
C04205=1039.135,328.941,378.214,172.169,43.122,158.336
C04206=1039.127,328.693,378.250,172.164,43.120,158.335
C04207=1039.120,328.446,378.285,172.159,43.117,158.334
C04208=1039.112,328.198,378.320,172.155,43.115,158.333
C04209=1039.105,327.951,378.355,172.149,43.113,158.332
C04210=1039.098,327.704,378.390,172.144,43.110,158.331
C04211=1039.090,327.456,378.426,172.140,43.108,158.330
C04212=1039.083,327.209,378.460,172.135,43.106,158.329
C04213=1039.075,326.961,378.496,172.130,43.104,158.329
C04214=1039.068,326.714,378.531,172.126,43.101,158.328
C04215=1039.061,326.467,378.566,172.121,43.099,158.327
C04216=1039.054,326.219,378.601,172.117,43.097,158.326
C04217=1039.046,325.972,378.636,172.112,43.095,158.325
C04218=1039.039,325.724,378.671,172.107,43.093,158.324
C04219=1039.031,325.477,378.706,172.103,43.090,158.323
C04220=1039.024,325.229,378.741,172.098,43.088,158.322
C04221=1039.017,324.982,378.775,172.094,43.086,158.322
C04222=1039.010,324.734,378.811,172.089,43.084,158.321
C04223=1039.002,324.487,378.845,172.084,43.081,158.320
C04224=1038.995,324.240,378.881,172.080,43.079,158.319
C04225=1038.988,323.993,378.915,172.074,43.077,158.318
C04226=1038.980,323.745,378.951,172.070,43.075,158.317
C04227=1038.974,323.497,378.985,172.065,43.073,158.316
C04228=1038.966,323.250,379.020,172.061,43.071,158.316
C04229=1038.960,323.002,379.055,172.056,43.068,158.315
C04230=1038.952,322.755,379.089,172.052,43.066,158.314
C04231=1038.945,322.507,379.125,172.047,43.064,158.313
C04232=1038.937,322.260,379.159,172.043,43.062,158.312
C04233=1038.931,322.012,379.194,172.038,43.060,158.311
C04234=1038.923,321.765,379.228,172.034,43.057,158.310
C04235=1038.917,321.518,379.263,172.029,43.055,158.309
C04236=1038.909,321.271,379.298,172.025,43.053,158.309
C04237=1038.902,321.022,379.333,172.020,43.051,158.308
C04238=1038.894,320.775,379.367,172.016,43.049,158.307
C04239=1038.884,320.415,379.417,172.010,43.046,158.306
C04240=1038.874,320.054,379.468,172.003,43.042,158.305
C04241=1038.864,319.694,379.518,171.997,43.040,158.303
C04242=1038.854,319.333,379.569,171.990,43.036,158.302
C04243=1038.847,319.086,379.603,171.985,43.034,158.301
C04244=1038.840,318.838,379.638,171.981,43.032,158.301
C04245=1038.833,318.591,379.672,171.976,43.030,158.300
C04246=1038.826,318.343,379.707,171.972,43.028,158.299
C04247=1038.819,318.096,379.741,171.967,43.026,158.298
C04248=1038.812,317.848,379.775,171.963,43.024,158.297
C04249=1038.805,317.601,379.810,171.959,43.022,158.297
C04250=1038.798,317.353,379.844,171.954,43.020,158.296
C04251=1038.791,317.106,379.879,171.950,43.017,158.295
C04252=1038.783,316.859,379.913,171.945,43.016,158.294
C04253=1038.777,316.611,379.948,171.941,43.013,158.293
C04254=1038.769,316.363,379.982,171.937,43.011,158.293
C04255=1038.763,316.116,380.017,171.932,43.009,158.292
C04256=1038.756,315.868,380.051,171.928,43.007,158.291
C04257=1038.749,315.620,380.085,171.925,43.005,158.290
C04258=1038.742,315.374,380.119,171.919,43.003,158.289
C04259=1038.736,315.126,380.154,171.916,43.001,158.288
C04260=1038.728,314.878,380.188,171.911,42.999,158.288
C04261=1038.722,314.630,380.222,171.907,42.997,158.287
C04262=1038.715,314.383,380.257,171.903,42.995,158.286
C04263=1038.707,314.136,380.290,171.898,42.993,158.285
C04264=1038.701,313.888,380.325,171.894,42.991,158.284
C04265=1038.694,313.641,380.358,171.890,42.989,158.284
C04266=1038.688,313.393,380.393,171.885,42.987,158.283
C04267=1038.680,313.146,380.427,171.881,42.985,158.282
C04268=1038.674,312.898,380.462,171.877,42.983,158.281
C04269=1038.667,312.651,380.495,171.872,42.981,158.281
C04270=1038.660,312.403,380.529,171.868,42.979,158.280
C04271=1038.653,312.156,380.564,171.864,42.976,158.279
C04272=1038.646,311.908,380.598,171.860,42.975,158.278
C04273=1038.639,311.660,380.632,171.855,42.973,158.278
C04274=1038.633,311.413,380.664,171.851,42.971,158.277
C04275=1038.625,311.165,380.698,171.847,42.969,158.276
C04276=1038.618,310.917,380.732,171.843,42.967,158.275
C04277=1038.610,310.670,380.765,171.839,42.965,158.275
C04278=1038.603,310.422,380.799,171.834,42.964,158.274
C04279=1038.596,310.175,380.833,171.830,42.962,158.273
C04280=1038.589,309.928,380.866,171.826,42.960,158.272
C04281=1038.582,309.679,380.900,171.821,42.958,158.272
C04282=1038.575,309.432,380.933,171.817,42.956,158.271
C04283=1038.567,309.184,380.967,171.814,42.954,158.270
C04284=1038.560,308.937,381.000,171.809,42.953,158.269
C04285=1038.554,308.689,381.033,171.805,42.951,158.269
C04286=1038.547,308.441,381.067,171.801,42.949,158.268
C04287=1038.539,308.194,381.101,171.797,42.947,158.267
C04288=1038.533,307.947,381.134,171.792,42.946,158.267
C04289=1038.525,307.699,381.167,171.789,42.944,158.266
C04290=1038.518,307.451,381.201,171.785,42.942,158.265
C04291=1038.511,307.204,381.234,171.780,42.940,158.264
C04292=1038.504,306.956,381.267,171.776,42.938,158.264
C04293=1038.497,306.708,381.301,171.772,42.936,158.263
C04294=1038.490,306.460,381.334,171.768,42.935,158.262
C04295=1038.480,306.105,381.382,171.762,42.932,158.261
C04296=1038.470,305.750,381.430,171.756,42.930,158.260
C04297=1038.460,305.394,381.477,171.751,42.927,158.259
C04298=1038.450,305.038,381.525,171.745,42.925,158.258
C04299=1038.443,304.790,381.558,171.741,42.923,158.258
C04300=1038.436,304.543,381.591,171.736,42.921,158.257
C04301=1038.429,304.295,381.624,171.732,42.919,158.256
C04302=1038.423,304.048,381.658,171.728,42.917,158.255
C04303=1038.416,303.800,381.691,171.724,42.916,158.255
C04304=1038.409,303.553,381.724,171.720,42.914,158.254
C04305=1038.401,303.305,381.757,171.716,42.912,158.253
C04306=1038.395,303.058,381.790,171.712,42.911,158.253
C04307=1038.388,302.810,381.823,171.708,42.909,158.252
C04308=1038.381,302.561,381.857,171.704,42.907,158.251
C04309=1038.374,302.315,381.889,171.700,42.905,158.251
C04310=1038.367,302.066,381.923,171.695,42.904,158.250
C04311=1038.360,301.819,381.955,171.692,42.902,158.249
C04312=1038.353,301.571,381.989,171.688,42.900,158.249
C04313=1038.347,301.323,382.022,171.684,42.899,158.248
C04314=1038.340,301.076,382.054,171.680,42.897,158.247
C04315=1038.333,300.828,382.088,171.676,42.895,158.247
C04316=1038.326,300.581,382.121,171.673,42.893,158.246
C04317=1038.320,300.333,382.154,171.668,42.892,158.245
C04318=1038.313,300.085,382.186,171.664,42.890,158.245
C04319=1038.306,299.837,382.219,171.660,42.888,158.244
C04320=1038.299,299.590,382.252,171.656,42.886,158.243
C04321=1038.292,299.342,382.286,171.653,42.885,158.243
C04322=1038.286,299.094,382.318,171.649,42.883,158.242
C04323=1038.279,298.847,382.350,171.645,42.881,158.241
C04324=1038.272,298.599,382.384,171.641,42.880,158.241
C04325=1038.266,298.351,382.416,171.636,42.878,158.240
C04326=1038.259,298.104,382.450,171.633,42.877,158.239
C04327=1038.251,297.856,382.482,171.629,42.875,158.238
C04328=1038.245,297.608,382.515,171.625,42.873,158.238
C04329=1038.238,297.360,382.548,171.621,42.872,158.237
C04330=1038.232,297.113,382.581,171.617,42.870,158.236
C04331=1038.225,296.865,382.613,171.614,42.868,158.236
C04332=1038.219,296.618,382.646,171.610,42.867,158.235
C04333=1038.212,296.369,382.679,171.606,42.865,158.234
C04334=1038.205,296.122,382.712,171.602,42.863,158.234
C04335=1038.198,295.874,382.744,171.599,42.861,158.233
C04336=1038.191,295.626,382.777,171.595,42.860,158.233
C04337=1038.185,295.379,382.810,171.591,42.858,158.232
C04338=1038.179,295.131,382.842,171.587,42.857,158.231
C04339=1038.172,294.882,382.874,171.583,42.855,158.231
C04340=1038.165,294.635,382.906,171.579,42.854,158.230
C04341=1038.158,294.388,382.939,171.575,42.852,158.229
C04342=1038.151,294.140,382.971,171.571,42.850,158.229
C04343=1038.144,293.892,383.004,171.568,42.849,158.228
C04344=1038.138,293.644,383.036,171.564,42.847,158.227
C04345=1038.131,293.396,383.068,171.560,42.846,158.227
C04346=1038.124,293.148,383.101,171.556,42.844,158.226
C04347=1038.117,292.901,383.132,171.553,42.843,158.226
C04348=1038.111,292.653,383.165,171.549,42.841,158.225
C04349=1038.103,292.405,383.198,171.545,42.839,158.224
C04350=1038.096,292.157,383.229,171.541,42.838,158.224
C04351=1038.087,291.818,383.273,171.537,42.836,158.223
C04352=1038.078,291.479,383.318,171.531,42.834,158.222
C04353=1038.068,291.140,383.361,171.526,42.832,158.221
C04354=1038.059,290.802,383.405,171.521,42.830,158.220
C04355=1038.052,290.554,383.437,171.517,42.829,158.220
C04356=1038.046,290.306,383.469,171.513,42.827,158.219
C04357=1038.039,290.059,383.502,171.509,42.825,158.219
C04358=1038.032,289.811,383.533,171.506,42.824,158.218
C04359=1038.026,289.563,383.566,171.502,42.823,158.217
C04360=1038.018,289.315,383.598,171.498,42.821,158.217
C04361=1038.012,289.067,383.629,171.495,42.819,158.216
C04362=1038.005,288.819,383.661,171.491,42.818,158.216
C04363=1037.998,288.572,383.693,171.487,42.817,158.215
C04364=1037.991,288.324,383.725,171.484,42.815,158.214
C04365=1037.984,288.075,383.757,171.480,42.814,158.214
C04366=1037.977,287.827,383.789,171.476,42.812,158.213
C04367=1037.970,287.580,383.821,171.472,42.811,158.213
C04368=1037.964,287.332,383.853,171.469,42.809,158.212
C04369=1037.958,287.084,383.884,171.465,42.808,158.211
C04370=1037.951,286.837,383.916,171.461,42.807,158.211
C04371=1037.944,286.589,383.948,171.459,42.805,158.210
C04372=1037.937,286.341,383.979,171.455,42.804,158.210
C04373=1037.930,286.092,384.011,171.451,42.802,158.209
C04374=1037.923,285.845,384.043,171.448,42.801,158.209
C04375=1037.916,285.597,384.075,171.444,42.799,158.208
C04376=1037.909,285.349,384.106,171.440,42.798,158.207
C04377=1037.903,285.101,384.137,171.437,42.797,158.207
C04378=1037.896,284.853,384.169,171.433,42.795,158.206
C04379=1037.889,284.606,384.200,171.429,42.794,158.206
C04380=1037.883,284.358,384.232,171.426,42.793,158.205
C04381=1037.875,284.110,384.264,171.422,42.791,158.205
C04382=1037.869,283.862,384.295,171.418,42.790,158.204
C04383=1037.861,283.614,384.327,171.415,42.789,158.203
C04384=1037.855,283.366,384.358,171.411,42.787,158.203
C04385=1037.848,283.118,384.390,171.407,42.786,158.202
C04386=1037.841,282.870,384.421,171.404,42.785,158.202
C04387=1037.835,282.622,384.453,171.400,42.783,158.201
C04388=1037.828,282.374,384.484,171.398,42.782,158.201
C04389=1037.821,282.126,384.516,171.394,42.780,158.200
C04390=1037.814,281.879,384.547,171.390,42.779,158.200
C04391=1037.808,281.631,384.579,171.387,42.778,158.199
C04392=1037.801,281.383,384.610,171.383,42.776,158.198
C04393=1037.794,281.135,384.641,171.379,42.775,158.198
C04394=1037.787,280.887,384.673,171.376,42.774,158.197
C04395=1037.781,280.639,384.704,171.372,42.772,158.197
C04396=1037.774,280.391,384.736,171.369,42.771,158.196
C04397=1037.768,280.143,384.766,171.366,42.770,158.196
C04398=1037.761,279.895,384.798,171.362,42.768,158.195
C04399=1037.755,279.647,384.829,171.358,42.767,158.195
C04400=1037.748,279.400,384.860,171.355,42.766,158.194
C04401=1037.741,279.152,384.891,171.351,42.764,158.193
C04402=1037.734,278.904,384.923,171.347,42.763,158.193
C04403=1037.727,278.656,384.954,171.345,42.761,158.192
C04404=1037.721,278.408,384.985,171.341,42.760,158.192
C04405=1037.714,278.160,385.016,171.338,42.759,158.191
C04406=1037.707,277.912,385.048,171.334,42.758,158.191
C04407=1037.698,277.585,385.089,171.329,42.756,158.190
C04408=1037.690,277.258,385.129,171.324,42.754,158.189
C04409=1037.681,276.931,385.170,171.321,42.753,158.189
C04410=1037.672,276.604,385.211,171.316,42.751,158.188
C04411=1037.664,276.356,385.242,171.312,42.750,158.187
C04412=1037.658,276.108,385.273,171.308,42.749,158.187
C04413=1037.651,275.860,385.304,171.306,42.747,158.186
C04414=1037.644,275.612,385.334,171.302,42.746,158.186
C04415=1037.637,275.364,385.365,171.299,42.745,158.185
C04416=1037.631,275.117,385.397,171.295,42.744,158.185
C04417=1037.625,274.868,385.427,171.291,42.742,158.184
C04418=1037.617,274.620,385.458,171.289,42.741,158.184
C04419=1037.611,274.372,385.489,171.285,42.740,158.183
C04420=1037.604,274.124,385.520,171.282,42.739,158.183
C04421=1037.597,273.876,385.550,171.278,42.737,158.182
C04422=1037.590,273.628,385.582,171.275,42.737,158.182
C04423=1037.585,273.380,385.612,171.272,42.735,158.181
C04424=1037.577,273.132,385.643,171.268,42.734,158.181
C04425=1037.571,272.884,385.674,171.265,42.732,158.180
C04426=1037.564,272.636,385.704,171.261,42.732,158.180
C04427=1037.557,272.388,385.735,171.258,42.730,158.179
C04428=1037.551,272.140,385.766,171.255,42.729,158.179
C04429=1037.544,271.892,385.796,171.251,42.727,158.178
C04430=1037.537,271.644,385.827,171.248,42.727,158.178
C04431=1037.531,271.395,385.858,171.244,42.725,158.177
C04432=1037.524,271.149,385.888,171.242,42.724,158.177
C04433=1037.517,270.900,385.919,171.238,42.723,158.176
C04434=1037.510,270.652,385.949,171.234,42.722,158.176
C04435=1037.504,270.403,385.980,171.231,42.720,158.175
C04436=1037.497,270.156,386.010,171.228,42.720,158.175
C04437=1037.491,269.908,386.041,171.225,42.718,158.174
C04438=1037.483,269.660,386.071,171.221,42.717,158.174
C04439=1037.477,269.411,386.102,171.218,42.716,158.173
C04440=1037.470,269.164,386.132,171.215,42.715,158.173
C04441=1037.463,268.916,386.163,171.212,42.714,158.172
C04442=1037.457,268.667,386.193,171.208,42.712,158.172
C04443=1037.449,268.419,386.223,171.204,42.711,158.171
C04444=1037.444,268.171,386.254,171.202,42.710,158.171
C04445=1037.436,267.923,386.284,171.198,42.709,158.170
C04446=1037.430,267.675,386.315,171.195,42.708,158.170
C04447=1037.423,267.428,386.345,171.192,42.707,158.169
C04448=1037.417,267.179,386.376,171.189,42.705,158.169
C04449=1037.410,266.931,386.406,171.185,42.705,158.168
C04450=1037.403,266.684,386.436,171.181,42.703,158.168
C04451=1037.397,266.435,386.466,171.179,42.702,158.167
C04452=1037.389,266.187,386.496,171.175,42.701,158.167
C04453=1037.382,265.939,386.527,171.172,42.700,158.166
C04454=1037.376,265.691,386.556,171.169,42.699,158.166
C04455=1037.369,265.443,386.587,171.166,42.698,158.165
C04456=1037.362,265.194,386.617,171.162,42.697,158.165
C04457=1037.356,264.947,386.647,171.160,42.696,158.165
C04458=1037.349,264.698,386.678,171.156,42.694,158.164
C04459=1037.343,264.451,386.707,171.153,42.694,158.164
C04460=1037.335,264.203,386.738,171.150,42.692,158.163
C04461=1037.329,263.953,386.768,171.147,42.691,158.163
C04462=1037.323,263.706,386.797,171.143,42.690,158.162
C04463=1037.313,263.384,386.836,171.139,42.689,158.162
C04464=1037.305,263.061,386.876,171.135,42.687,158.161
C04465=1037.297,262.739,386.915,171.131,42.686,158.160
C04466=1037.287,262.417,386.954,171.126,42.684,158.160
C04467=1037.281,262.168,386.984,171.124,42.683,158.159
C04468=1037.275,261.920,387.014,171.120,42.682,158.159
C04469=1037.268,261.672,387.044,171.117,42.681,158.158
C04470=1037.261,261.425,387.073,171.114,42.680,158.158
C04471=1037.254,261.176,387.103,171.111,42.679,158.157
C04472=1037.247,260.928,387.133,171.107,42.678,158.157
C04473=1037.241,260.680,387.163,171.105,42.677,158.157
C04474=1037.234,260.431,387.192,171.101,42.676,158.156
C04475=1037.226,260.184,387.221,171.098,42.675,158.156
C04476=1037.220,259.935,387.251,171.095,42.674,158.155
C04477=1037.212,259.687,387.281,171.092,42.674,158.155
C04478=1037.206,259.439,387.311,171.088,42.672,158.154
C04479=1037.199,259.191,387.340,171.086,42.671,158.154
C04480=1037.192,258.943,387.370,171.082,42.670,158.154
C04481=1037.186,258.694,387.399,171.080,42.669,158.153
C04482=1037.178,258.446,387.429,171.076,42.668,158.153
C04483=1037.172,258.198,387.458,171.073,42.667,158.152
C04484=1037.165,257.950,387.488,171.070,42.667,158.152
C04485=1037.158,257.702,387.517,171.067,42.665,158.151
C04486=1037.151,257.454,387.547,171.063,42.664,158.151
C04487=1037.145,257.206,387.576,171.061,42.664,158.150
C04488=1037.137,256.957,387.606,171.057,42.662,158.150
C04489=1037.131,256.709,387.635,171.055,42.661,158.150
C04490=1037.124,256.461,387.665,171.051,42.661,158.149
C04491=1037.118,256.213,387.694,171.048,42.660,158.149
C04492=1037.111,255.964,387.724,171.045,42.658,158.148
C04493=1037.104,255.716,387.754,171.042,42.657,158.148
C04494=1037.097,255.468,387.782,171.039,42.657,158.147
C04495=1037.090,255.220,387.812,171.036,42.656,158.147
C04496=1037.083,254.972,387.842,171.032,42.654,158.146
C04497=1037.077,254.723,387.871,171.030,42.654,158.146
C04498=1037.071,254.476,387.900,171.026,42.653,158.146
C04499=1037.064,254.227,387.930,171.024,42.652,158.145
C04500=1037.057,253.979,387.959,171.020,42.651,158.145
C04501=1037.050,253.731,387.989,171.018,42.650,158.144
C04502=1037.043,253.483,388.017,171.014,42.649,158.144
C04503=1037.036,253.234,388.047,171.012,42.648,158.144
C04504=1037.030,252.987,388.076,171.008,42.647,158.143
C04505=1037.024,252.738,388.106,171.005,42.646,158.143
C04506=1037.017,252.490,388.135,171.003,42.645,158.142
C04507=1037.011,252.242,388.164,170.999,42.644,158.142
C04508=1037.003,251.993,388.194,170.996,42.643,158.141
C04509=1036.997,251.745,388.223,170.993,42.642,158.141
C04510=1036.990,251.497,388.252,170.991,42.641,158.141
C04511=1036.983,251.249,388.281,170.987,42.640,158.140
C04512=1036.977,251.001,388.311,170.985,42.639,158.140
C04513=1036.971,250.753,388.340,170.981,42.638,158.139
C04514=1036.964,250.504,388.369,170.979,42.637,158.139
C04515=1036.957,250.256,388.398,170.975,42.636,158.138
C04516=1036.951,250.008,388.427,170.973,42.635,158.138
C04517=1036.944,249.759,388.456,170.969,42.634,158.138
C04518=1036.937,249.511,388.485,170.967,42.633,158.137
C04519=1036.929,249.187,388.524,170.963,42.632,158.137
C04520=1036.920,248.864,388.562,170.958,42.630,158.136
C04521=1036.912,248.539,388.600,170.955,42.629,158.135
C04522=1036.903,248.216,388.637,170.951,42.628,158.135
C04523=1036.897,247.968,388.666,170.948,42.627,158.135
C04524=1036.890,247.719,388.696,170.945,42.626,158.134
C04525=1036.884,247.471,388.725,170.942,42.625,158.134
C04526=1036.877,247.223,388.754,170.939,42.624,158.133
C04527=1036.870,246.975,388.782,170.937,42.623,158.133
C04528=1036.864,246.726,388.812,170.933,42.622,158.132
C04529=1036.857,246.478,388.841,170.931,42.621,158.132
C04530=1036.851,246.230,388.870,170.927,42.620,158.132
C04531=1036.845,245.982,388.899,170.925,42.619,158.131
C04532=1036.838,245.734,388.927,170.921,42.618,158.131
C04533=1036.831,245.485,388.957,170.919,42.617,158.130
C04534=1036.825,245.237,388.986,170.917,42.616,158.130
C04535=1036.818,244.989,389.015,170.913,42.616,158.130
C04536=1036.812,244.741,389.044,170.911,42.615,158.129
C04537=1036.805,244.492,389.073,170.907,42.613,158.129
C04538=1036.798,244.244,389.102,170.905,42.612,158.128
C04539=1036.791,243.997,389.130,170.901,42.612,158.128
C04540=1036.785,243.748,389.158,170.899,42.611,158.128
C04541=1036.778,243.500,389.187,170.895,42.610,158.127
C04542=1036.772,243.251,389.216,170.893,42.609,158.127
C04543=1036.765,243.003,389.245,170.890,42.608,158.126
C04544=1036.759,242.755,389.273,170.887,42.607,158.126
C04545=1036.752,242.506,389.302,170.885,42.606,158.126
C04546=1036.745,242.259,389.331,170.881,42.606,158.125
C04547=1036.739,242.010,389.360,170.879,42.605,158.125
C04548=1036.732,241.761,389.388,170.876,42.603,158.124
C04549=1036.726,241.513,389.417,170.873,42.602,158.124
C04550=1036.719,241.265,389.445,170.870,42.601,158.124
C04551=1036.712,241.017,389.474,170.867,42.601,158.123
C04552=1036.706,240.768,389.503,170.864,42.600,158.123
C04553=1036.699,240.520,389.531,170.862,42.599,158.122
C04554=1036.692,240.271,389.559,170.859,42.598,158.122
C04555=1036.686,240.023,389.588,170.856,42.597,158.122
C04556=1036.679,239.776,389.617,170.853,42.596,158.121
C04557=1036.672,239.527,389.644,170.850,42.595,158.121
C04558=1036.666,239.279,389.673,170.848,42.595,158.120
C04559=1036.659,239.030,389.701,170.844,42.594,158.120
C04560=1036.652,238.782,389.730,170.842,42.593,158.120
C04561=1036.645,238.534,389.758,170.839,42.592,158.119
C04562=1036.639,238.285,389.787,170.836,42.591,158.119
C04563=1036.632,238.037,389.814,170.834,42.590,158.119
C04564=1036.625,237.789,389.843,170.830,42.589,158.118
C04565=1036.619,237.540,389.871,170.828,42.589,158.118
C04566=1036.612,237.292,389.900,170.825,42.588,158.118
C04567=1036.605,237.043,389.928,170.822,42.588,158.117
C04568=1036.598,236.796,389.956,170.820,42.587,158.117
C04569=1036.592,236.547,389.985,170.816,42.586,158.116
C04570=1036.585,236.298,390.012,170.814,42.585,158.116
C04571=1036.578,236.051,390.041,170.811,42.584,158.116
C04572=1036.572,235.802,390.068,170.808,42.583,158.115
C04573=1036.565,235.554,390.097,170.806,42.582,158.115
C04574=1036.559,235.306,390.125,170.803,42.581,158.115
C04575=1036.550,234.976,390.163,170.799,42.580,158.114
C04576=1036.540,234.646,390.200,170.795,42.579,158.114
C04577=1036.532,234.317,390.237,170.791,42.578,158.113
C04578=1036.523,233.986,390.274,170.788,42.577,158.113
C04579=1036.516,233.739,390.303,170.786,42.576,158.112
C04580=1036.509,233.490,390.331,170.782,42.576,158.112
C04581=1036.504,233.241,390.359,170.780,42.575,158.111
C04582=1036.497,232.994,390.387,170.777,42.574,158.111
C04583=1036.490,232.745,390.415,170.775,42.573,158.111
C04584=1036.483,232.497,390.443,170.771,42.572,158.110
C04585=1036.476,232.248,390.471,170.769,42.571,158.110
C04586=1036.470,232.000,390.500,170.767,42.570,158.110
C04587=1036.464,231.752,390.527,170.763,42.569,158.109
C04588=1036.457,231.503,390.555,170.761,42.568,158.109
C04589=1036.450,231.255,390.583,170.759,42.568,158.109
C04590=1036.444,231.006,390.611,170.755,42.567,158.108
C04591=1036.437,230.759,390.639,170.753,42.566,158.108
C04592=1036.430,230.510,390.667,170.750,42.566,158.107
C04593=1036.423,230.262,390.694,170.747,42.565,158.107
C04594=1036.417,230.013,390.723,170.744,42.564,158.107
C04595=1036.411,229.764,390.751,170.742,42.563,158.106
C04596=1036.404,229.516,390.778,170.740,42.562,158.106
C04597=1036.397,229.268,390.806,170.736,42.562,158.106
C04598=1036.391,229.019,390.834,170.734,42.561,158.105
C04599=1036.384,228.771,390.861,170.731,42.560,158.105
C04600=1036.377,228.523,390.890,170.729,42.559,158.105
C04601=1036.371,228.275,390.917,170.726,42.558,158.104
C04602=1036.364,228.027,390.945,170.723,42.557,158.104
C04603=1036.357,227.778,390.973,170.721,42.556,158.103
C04604=1036.351,227.530,391.000,170.718,42.556,158.103
C04605=1036.344,227.281,391.027,170.715,42.555,158.103
C04606=1036.337,227.033,391.055,170.713,42.554,158.102
C04607=1036.330,226.784,391.082,170.710,42.553,158.102
C04608=1036.324,226.536,391.110,170.707,42.553,158.102
C04609=1036.317,226.287,391.138,170.705,42.552,158.101
C04610=1036.310,226.039,391.166,170.702,42.551,158.101
C04611=1036.304,225.790,391.193,170.700,42.551,158.101
C04612=1036.296,225.542,391.220,170.697,42.550,158.100
C04613=1036.289,225.294,391.248,170.694,42.549,158.100
C04614=1036.283,225.045,391.276,170.692,42.549,158.100
C04615=1036.276,224.796,391.303,170.689,42.548,158.099
C04616=1036.270,224.548,391.331,170.686,42.547,158.099
C04617=1036.264,224.300,391.358,170.684,42.547,158.099
C04618=1036.256,224.052,391.385,170.681,42.546,158.098
C04619=1036.249,223.804,391.413,170.679,42.545,158.098
C04620=1036.243,223.555,391.441,170.675,42.544,158.098
C04621=1036.236,223.306,391.468,170.673,42.544,158.097
C04622=1036.230,223.058,391.495,170.671,42.543,158.097
C04623=1036.223,222.809,391.523,170.668,42.542,158.097
C04624=1036.216,222.561,391.550,170.665,42.541,158.096
C04625=1036.210,222.313,391.578,170.662,42.540,158.096
C04626=1036.203,222.064,391.605,170.660,42.540,158.096
C04627=1036.197,221.816,391.632,170.658,42.539,158.095
C04628=1036.190,221.567,391.660,170.655,42.538,158.095
C04629=1036.182,221.319,391.687,170.653,42.537,158.095
C04630=1036.176,221.070,391.714,170.649,42.536,158.094
C04631=1036.168,220.734,391.751,170.646,42.535,158.094
C04632=1036.159,220.397,391.789,170.643,42.535,158.093
C04633=1036.150,220.060,391.826,170.639,42.533,158.093
C04634=1036.141,219.722,391.863,170.636,42.532,158.092
C04635=1036.134,219.474,391.890,170.633,42.531,158.092
C04636=1036.127,219.225,391.917,170.631,42.531,158.092
C04637=1036.120,218.977,391.944,170.628,42.530,158.091
C04638=1036.114,218.728,391.970,170.626,42.529,158.091
C04639=1036.107,218.480,391.998,170.624,42.528,158.091
C04640=1036.100,218.232,392.025,170.620,42.528,158.090
C04641=1036.093,217.983,392.052,170.618,42.527,158.090
C04642=1036.086,217.735,392.079,170.616,42.526,158.090
C04643=1036.080,217.486,392.106,170.613,42.526,158.089
C04644=1036.073,217.238,392.133,170.611,42.525,158.089
C04645=1036.066,216.989,392.160,170.607,42.524,158.089
C04646=1036.059,216.741,392.187,170.605,42.524,158.088
C04647=1036.053,216.492,392.214,170.603,42.523,158.088
C04648=1036.046,216.244,392.241,170.600,42.522,158.088
C04649=1036.040,215.995,392.268,170.598,42.522,158.088
C04650=1036.032,215.747,392.295,170.596,42.521,158.087
C04651=1036.026,215.498,392.322,170.593,42.520,158.087
C04652=1036.019,215.250,392.348,170.590,42.520,158.087
C04653=1036.013,215.002,392.376,170.588,42.519,158.086
C04654=1036.006,214.753,392.403,170.585,42.518,158.086
C04655=1035.999,214.505,392.430,170.583,42.518,158.086
C04656=1035.993,214.256,392.457,170.581,42.517,158.085
C04657=1035.986,214.007,392.483,170.578,42.516,158.085
C04658=1035.979,213.759,392.511,170.576,42.515,158.085
C04659=1035.973,213.511,392.537,170.573,42.515,158.084
C04660=1035.966,213.262,392.564,170.570,42.514,158.084
C04661=1035.959,213.014,392.591,170.568,42.513,158.084
C04662=1035.953,212.765,392.618,170.565,42.512,158.083
C04663=1035.946,212.517,392.644,170.563,42.512,158.083
C04664=1035.939,212.268,392.672,170.561,42.511,158.083
C04665=1035.933,212.020,392.698,170.558,42.510,158.082
C04666=1035.926,211.771,392.725,170.556,42.509,158.082
C04667=1035.919,211.523,392.752,170.554,42.508,158.082
C04668=1035.913,211.275,392.779,170.551,42.508,158.081
C04669=1035.906,211.026,392.805,170.548,42.507,158.081
C04670=1035.899,210.777,392.832,170.546,42.506,158.081
C04671=1035.893,210.529,392.859,170.543,42.506,158.080
C04672=1035.886,210.281,392.886,170.541,42.505,158.080
C04673=1035.879,210.032,392.912,170.538,42.504,158.080
C04674=1035.873,209.783,392.939,170.536,42.504,158.079
C04675=1035.866,209.535,392.965,170.534,42.503,158.079
C04676=1035.859,209.286,392.993,170.532,42.503,158.079
C04677=1035.853,209.038,393.019,170.529,42.502,158.078
C04678=1035.845,208.789,393.045,170.527,42.501,158.078
C04679=1035.838,208.541,393.072,170.525,42.500,158.078
C04680=1035.833,208.292,393.098,170.522,42.499,158.078
C04681=1035.825,208.044,393.125,170.519,42.499,158.077
C04682=1035.819,207.796,393.151,170.516,42.498,158.077
C04683=1035.812,207.547,393.177,170.514,42.497,158.077
C04684=1035.805,207.298,393.205,170.512,42.497,158.076
C04685=1035.799,207.050,393.231,170.509,42.496,158.076
C04686=1035.792,206.802,393.257,170.507,42.496,158.076
C04687=1035.783,206.470,393.293,170.504,42.494,158.075
C04688=1035.774,206.139,393.328,170.501,42.494,158.075
C04689=1035.764,205.807,393.363,170.498,42.493,158.074
C04690=1035.756,205.475,393.398,170.494,42.492,158.074
C04691=1035.729,204.425,393.504,170.178,42.388,158.031
C04692=1035.723,204.176,393.529,170.173,42.388,158.030
C04693=1035.718,203.928,393.554,170.170,42.388,158.030
C04694=1035.711,203.680,393.579,170.167,42.388,158.030
C04695=1035.705,203.431,393.605,170.164,42.388,158.030
C04696=1035.699,203.182,393.629,170.161,42.388,158.030
C04697=1035.693,202.933,393.655,170.158,42.388,158.029
C04698=1035.686,202.685,393.679,170.154,42.388,158.029
C04699=1035.680,202.436,393.705,170.150,42.388,158.029
C04700=1035.675,202.187,393.729,170.147,42.388,158.029
C04701=1035.668,201.939,393.754,170.144,42.388,158.029
C04702=1035.662,201.690,393.780,170.141,42.389,158.028
C04703=1035.656,201.441,393.805,170.138,42.389,158.028
C04704=1035.650,201.192,393.830,170.134,42.388,158.028
C04705=1035.645,200.944,393.855,170.131,42.389,158.028
C04706=1035.638,200.695,393.879,170.128,42.389,158.028
C04707=1035.632,200.447,393.904,170.124,42.389,158.027
C04708=1035.626,200.198,393.929,170.121,42.389,158.027
C04709=1035.619,199.949,393.953,170.118,42.390,158.027
C04710=1035.613,199.701,393.978,170.115,42.390,158.027
C04711=1035.607,199.452,394.002,170.112,42.390,158.027
C04712=1035.600,199.203,394.028,170.108,42.390,158.027
C04713=1035.594,198.954,394.052,170.105,42.390,158.026
C04714=1035.588,198.706,394.077,170.101,42.391,158.026
C04715=1035.582,198.457,394.101,170.098,42.391,158.026
C04716=1035.576,198.208,394.125,170.095,42.391,158.026
C04717=1035.569,197.959,394.151,170.092,42.392,158.026
C04718=1035.563,197.710,394.175,170.089,42.392,158.025
C04719=1035.557,197.462,394.200,170.086,42.392,158.025
C04720=1035.551,197.213,394.224,170.082,42.392,158.025
C04721=1035.544,196.965,394.249,170.079,42.392,158.025
C04722=1035.538,196.716,394.273,170.075,42.393,158.025
C04723=1035.532,196.467,394.298,170.072,42.393,158.025
C04724=1035.525,196.219,394.322,170.069,42.393,158.024
C04725=1035.520,195.970,394.347,170.066,42.394,158.024
C04726=1035.513,195.721,394.371,170.063,42.393,158.024
C04727=1035.507,195.473,394.396,170.060,42.394,158.024
C04728=1035.501,195.224,394.420,170.057,42.394,158.024
C04729=1035.495,194.974,394.444,170.053,42.394,158.024
C04730=1035.488,194.727,394.469,170.050,42.395,158.023
C04731=1035.483,194.477,394.493,170.047,42.395,158.023
C04732=1035.476,194.228,394.517,170.044,42.395,158.023
C04733=1035.470,193.981,394.542,170.041,42.395,158.023
C04734=1035.464,193.732,394.566,170.038,42.395,158.023
C04735=1035.458,193.482,394.591,170.034,42.396,158.023
C04736=1035.452,193.234,394.615,170.031,42.396,158.022
C04737=1035.446,192.985,394.640,170.028,42.396,158.022
C04738=1035.439,192.736,394.664,170.025,42.397,158.022
C04739=1035.434,192.488,394.688,170.021,42.397,158.022
C04740=1035.427,192.239,394.712,170.018,42.397,158.022
C04741=1035.422,191.990,394.737,170.015,42.397,158.022
C04742=1035.415,191.742,394.761,170.012,42.398,158.022
C04743=1035.409,191.493,394.786,170.009,42.398,158.021
C04744=1035.403,191.244,394.810,170.006,42.398,158.021
C04745=1035.397,190.995,394.834,170.003,42.399,158.021
C04746=1035.391,190.747,394.858,170.000,42.399,158.021
C04747=1035.385,190.497,394.882,169.997,42.399,158.021
C04748=1035.378,190.248,394.906,169.994,42.399,158.021
C04749=1035.373,190.000,394.931,169.991,42.400,158.020
C04750=1035.366,189.751,394.955,169.987,42.400,158.020
C04751=1035.361,189.503,394.980,169.984,42.400,158.020
C04752=1035.354,189.218,395.007,169.981,42.401,158.020
C04753=1035.347,188.935,395.035,169.977,42.401,158.020
C04754=1035.340,188.651,395.063,169.974,42.401,158.020
C04755=1035.333,188.366,395.090,169.970,42.402,158.019
C04756=1035.327,188.118,395.114,169.968,42.402,158.019
C04757=1035.321,187.869,395.138,169.965,42.402,158.019
C04758=1035.315,187.620,395.162,169.962,42.402,158.019
C04759=1035.309,187.371,395.186,169.959,42.403,158.019
C04760=1035.303,187.123,395.210,169.956,42.403,158.019
C04761=1035.297,186.873,395.235,169.952,42.403,158.019
C04762=1035.291,186.625,395.258,169.949,42.404,158.018
C04763=1035.285,186.376,395.283,169.946,42.404,158.018
C04764=1035.279,186.128,395.307,169.943,42.405,158.018
C04765=1035.273,185.878,395.331,169.940,42.404,158.018
C04766=1035.267,185.630,395.355,169.937,42.405,158.018
C04767=1035.262,185.381,395.379,169.934,42.405,158.018
C04768=1035.255,185.132,395.403,169.931,42.406,158.018
C04769=1035.249,184.884,395.427,169.928,42.406,158.017
C04770=1035.244,184.635,395.452,169.925,42.406,158.017
C04771=1035.238,184.386,395.474,169.922,42.407,158.017
C04772=1035.233,184.137,395.499,169.918,42.407,158.017
C04773=1035.226,183.888,395.523,169.916,42.407,158.017
C04774=1035.221,183.640,395.547,169.913,42.407,158.017
C04775=1035.214,183.391,395.571,169.910,42.408,158.017
C04776=1035.208,183.143,395.595,169.907,42.408,158.016
C04777=1035.202,182.893,395.618,169.904,42.409,158.016
C04778=1035.196,182.645,395.642,169.901,42.409,158.016
C04779=1035.189,182.396,395.666,169.898,42.409,158.016
C04780=1035.183,182.147,395.689,169.895,42.410,158.016
C04781=1035.177,181.898,395.713,169.892,42.410,158.016
C04782=1035.171,181.649,395.736,169.889,42.411,158.016
C04783=1035.164,181.401,395.759,169.886,42.411,158.016
C04784=1035.157,181.152,395.783,169.883,42.412,158.016
C04785=1035.152,180.903,395.806,169.880,42.413,158.016
C04786=1035.145,180.654,395.830,169.877,42.413,158.015
C04787=1035.139,180.405,395.853,169.874,42.414,158.015
C04788=1035.133,180.156,395.877,169.871,42.414,158.015
C04789=1035.127,179.907,395.900,169.868,42.415,158.015
C04790=1035.120,179.658,395.924,169.865,42.415,158.015
C04791=1035.114,179.410,395.946,169.862,42.416,158.015
C04792=1035.108,179.162,395.970,169.859,42.416,158.015
C04793=1035.101,178.912,395.993,169.856,42.417,158.015
C04794=1035.095,178.664,396.017,169.853,42.418,158.015
C04795=1035.089,178.414,396.040,169.850,42.418,158.015
C04796=1035.083,178.166,396.064,169.847,42.419,158.014
C04797=1035.077,177.917,396.087,169.845,42.419,158.014
C04798=1035.070,177.668,396.110,169.842,42.419,158.014
C04799=1035.064,177.419,396.133,169.839,42.420,158.014
C04800=1035.058,177.171,396.157,169.836,42.420,158.014
C04801=1035.052,176.921,396.180,169.833,42.421,158.014
C04802=1035.046,176.673,396.203,169.830,42.422,158.014
C04803=1035.040,176.424,396.226,169.827,42.422,158.014
C04804=1035.034,176.175,396.250,169.824,42.423,158.014
C04805=1035.027,175.927,396.273,169.821,42.423,158.014
C04806=1035.021,175.678,396.296,169.818,42.424,158.013
C04807=1035.015,175.428,396.319,169.815,42.424,158.013
C04808=1035.009,175.180,396.343,169.813,42.425,158.013
C04809=1035.003,174.931,396.366,169.810,42.426,158.013
C04810=1034.997,174.681,396.389,169.807,42.426,158.013
C04811=1034.990,174.433,396.412,169.804,42.427,158.013
C04812=1034.984,174.185,396.435,169.801,42.427,158.013
C04813=1034.979,173.936,396.458,169.798,42.428,158.013
C04814=1034.972,173.687,396.482,169.794,42.428,158.013
C04815=1034.966,173.438,396.505,169.791,42.429,158.013
C04816=1034.959,173.153,396.531,169.789,42.430,158.013
C04817=1034.952,172.869,396.558,169.786,42.430,158.013
C04818=1034.945,172.584,396.584,169.783,42.431,158.012
C04819=1034.938,172.300,396.610,169.778,42.431,158.012
C04820=1034.932,172.051,396.633,169.775,42.432,158.012
C04821=1034.926,171.802,396.656,169.774,42.433,158.012
C04822=1034.920,171.553,396.680,169.771,42.433,158.012
C04823=1034.914,171.305,396.703,169.768,42.434,158.012
C04824=1034.908,171.056,396.725,169.764,42.434,158.012
C04825=1034.902,170.806,396.749,169.761,42.435,158.012
C04826=1034.896,170.557,396.772,169.758,42.435,158.012
C04827=1034.890,170.309,396.795,169.757,42.436,158.012
C04828=1034.884,170.060,396.818,169.754,42.436,158.012
C04829=1034.878,169.812,396.841,169.750,42.437,158.012
C04830=1034.872,169.563,396.863,169.747,42.437,158.011
C04831=1034.866,169.313,396.887,169.744,42.438,158.011
C04832=1034.860,169.064,396.910,169.742,42.438,158.011
C04833=1034.854,168.815,396.933,169.740,42.439,158.011
C04834=1034.847,168.567,396.956,169.737,42.440,158.011
C04835=1034.842,168.319,396.979,169.733,42.440,158.011
C04836=1034.836,168.070,397.002,169.730,42.441,158.011
C04837=1034.830,167.821,397.025,169.728,42.441,158.011
C04838=1034.824,167.571,397.048,169.726,42.442,158.011
C04839=1034.817,167.323,397.070,169.723,42.443,158.011
C04840=1034.812,167.074,397.093,169.719,42.443,158.011
C04841=1034.806,166.825,397.116,169.716,42.443,158.010
C04842=1034.800,166.576,397.139,169.714,42.444,158.010
C04843=1034.794,166.327,397.162,169.711,42.444,158.010
C04844=1034.788,166.078,397.184,169.709,42.445,158.010
C04845=1034.782,165.830,397.207,169.705,42.446,158.010
C04846=1034.776,165.581,397.230,169.703,42.446,158.010
C04847=1034.771,165.332,397.253,169.700,42.447,158.010
C04848=1034.764,165.083,397.276,169.697,42.447,158.010
C04849=1034.758,164.834,397.299,169.695,42.448,158.010
C04850=1034.752,164.585,397.322,169.693,42.449,158.010
C04851=1034.746,164.336,397.345,169.689,42.449,158.010
C04852=1034.740,164.087,397.367,169.686,42.449,158.010
C04853=1034.734,163.838,397.390,169.683,42.450,158.010
C04854=1034.729,163.589,397.413,169.682,42.451,158.010
C04855=1034.723,163.340,397.436,169.679,42.451,158.009
C04856=1034.717,163.092,397.459,169.675,42.452,158.009
C04857=1034.711,162.842,397.481,169.672,42.452,158.009
C04858=1034.705,162.593,397.503,169.670,42.453,158.009
C04859=1034.699,162.345,397.526,169.668,42.454,158.009
C04860=1034.694,162.096,397.549,169.665,42.454,158.009
C04861=1034.687,161.847,397.572,169.661,42.455,158.009
C04862=1034.681,161.598,397.595,169.659,42.455,158.009
C04863=1034.676,161.349,397.618,169.656,42.455,158.009
C04864=1034.670,161.100,397.641,169.654,42.457,158.009
C04865=1034.664,160.851,397.662,169.652,42.457,158.009
C04866=1034.658,160.602,397.685,169.649,42.457,158.009
C04867=1034.652,160.353,397.708,169.645,42.458,158.008
C04868=1034.647,160.105,397.731,169.643,42.458,158.008
C04869=1034.640,159.856,397.753,169.641,42.459,158.008
C04870=1034.635,159.606,397.776,169.638,42.460,158.008
C04871=1034.628,159.358,397.798,169.635,42.461,158.008
C04872=1034.622,159.109,397.820,169.633,42.461,158.008
C04873=1034.616,158.860,397.843,169.630,42.462,158.008
C04874=1034.610,158.611,397.865,169.627,42.463,158.008
C04875=1034.604,158.362,397.887,169.624,42.463,158.008
C04876=1034.598,158.113,397.909,169.622,42.464,158.008
C04877=1034.592,157.864,397.932,169.619,42.465,158.008
C04878=1034.585,157.615,397.953,169.616,42.466,158.008
C04879=1034.580,157.366,397.976,169.613,42.466,158.008
C04880=1034.573,157.081,398.001,169.610,42.467,158.008
C04881=1034.566,156.797,398.027,169.607,42.468,158.008
C04882=1034.560,156.512,398.052,169.604,42.469,158.008
C04883=1034.552,156.227,398.078,169.601,42.469,158.008
C04884=1034.546,155.977,398.100,169.598,42.470,158.008
C04885=1034.540,155.729,398.122,169.595,42.471,158.008
C04886=1034.534,155.480,398.145,169.593,42.471,158.008
C04887=1034.528,155.231,398.167,169.590,42.472,158.008
C04888=1034.522,154.983,398.189,169.587,42.473,158.007
C04889=1034.516,154.733,398.211,169.586,42.474,158.008
C04890=1034.510,154.485,398.233,169.583,42.474,158.007
C04891=1034.504,154.236,398.255,169.580,42.475,158.007
C04892=1034.498,153.986,398.276,169.577,42.476,158.007
C04893=1034.492,153.737,398.299,169.575,42.477,158.007
C04894=1034.486,153.488,398.321,169.572,42.477,158.007
C04895=1034.479,153.240,398.343,169.569,42.478,158.007
C04896=1034.473,152.990,398.365,169.567,42.479,158.007
C04897=1034.467,152.741,398.387,169.564,42.480,158.007
C04898=1034.460,152.493,398.409,169.561,42.480,158.007
C04899=1034.455,152.243,398.431,169.558,42.481,158.007
C04900=1034.449,151.995,398.453,169.556,42.482,158.007
C04901=1034.443,151.746,398.475,169.553,42.483,158.007
C04902=1034.437,151.497,398.497,169.550,42.483,158.007
C04903=1034.430,151.248,398.519,169.548,42.484,158.007
C04904=1034.425,150.999,398.541,169.545,42.485,158.007
C04905=1034.419,150.749,398.563,169.543,42.486,158.007
C04906=1034.412,150.501,398.585,169.541,42.486,158.007
C04907=1034.407,150.252,398.606,169.538,42.487,158.007
C04908=1034.401,150.003,398.628,169.535,42.488,158.007
C04909=1034.394,149.754,398.650,169.533,42.489,158.007
C04910=1034.388,149.505,398.672,169.530,42.489,158.007
C04911=1034.382,149.256,398.694,169.527,42.490,158.007
C04912=1034.376,149.007,398.716,169.525,42.491,158.007
C04913=1034.370,148.757,398.737,169.522,42.492,158.007
C04914=1034.364,148.510,398.759,169.519,42.492,158.007
C04915=1034.358,148.260,398.781,169.517,42.493,158.007
C04916=1034.352,148.011,398.803,169.514,42.494,158.007
C04917=1034.346,147.762,398.824,169.511,42.495,158.007
C04918=1034.340,147.513,398.846,169.509,42.496,158.007
C04919=1034.334,147.265,398.868,169.506,42.496,158.006
C04920=1034.328,147.016,398.890,169.504,42.497,158.007
C04921=1034.321,146.766,398.911,169.502,42.498,158.006
C04922=1034.315,146.517,398.933,169.499,42.499,158.006
C04923=1034.309,146.268,398.955,169.496,42.500,158.006
C04924=1034.303,146.019,398.976,169.494,42.500,158.006
C04925=1034.297,145.770,398.997,169.491,42.501,158.006
C04926=1034.291,145.521,399.019,169.488,42.502,158.006
C04927=1034.285,145.272,399.041,169.486,42.503,158.006
C04928=1034.279,145.023,399.063,169.483,42.504,158.006
C04929=1034.272,144.774,399.085,169.480,42.504,158.006
C04930=1034.267,144.526,399.106,169.478,42.505,158.006
C04931=1034.261,144.276,399.128,169.476,42.506,158.006
C04932=1034.254,144.028,399.149,169.472,42.507,158.006
C04933=1034.248,143.778,399.170,169.471,42.508,158.006
C04934=1034.242,143.530,399.192,169.468,42.509,158.006
C04935=1034.236,143.281,399.213,169.465,42.509,158.006
C04936=1034.230,143.031,399.235,169.463,42.510,158.006
C04937=1034.224,142.782,399.256,169.460,42.511,158.006
C04938=1034.218,142.534,399.278,169.457,42.512,158.006
C04939=1034.212,142.285,399.299,169.455,42.513,158.006
C04940=1034.206,142.035,399.321,169.452,42.513,158.006
C04941=1034.200,141.786,399.343,169.450,42.514,158.006
C04942=1034.193,141.538,399.363,169.447,42.515,158.006
C04943=1034.187,141.288,399.384,169.444,42.516,158.006
C04944=1034.181,141.003,399.409,169.442,42.517,158.006
C04945=1034.173,140.718,399.434,169.439,42.518,158.006
C04946=1034.167,140.433,399.458,169.436,42.519,158.006
C04947=1034.159,140.147,399.483,169.433,42.520,158.006
C04948=1034.154,139.899,399.504,169.431,42.521,158.006
C04949=1034.148,139.649,399.525,169.428,42.521,158.006
C04950=1034.141,139.400,399.547,169.425,42.522,158.006
C04951=1034.136,139.152,399.568,169.423,42.523,158.006
C04952=1034.130,138.902,399.589,169.420,42.524,158.006
C04953=1034.123,138.653,399.610,169.418,42.525,158.006
C04954=1034.118,138.404,399.632,169.416,42.526,158.006
C04955=1034.111,138.155,399.653,169.413,42.526,158.006
C04956=1034.105,137.906,399.675,169.411,42.527,158.006
C04957=1034.099,137.657,399.695,169.408,42.528,158.006
C04958=1034.093,137.408,399.716,169.406,42.529,158.006
C04959=1034.087,137.159,399.738,169.403,42.530,158.006
C04960=1034.081,136.911,399.759,169.400,42.531,158.006
C04961=1034.075,136.661,399.780,169.398,42.532,158.006
C04962=1034.069,136.412,399.801,169.395,42.532,158.006
C04963=1034.062,136.163,399.822,169.392,42.533,158.006
C04964=1034.056,135.914,399.844,169.391,42.534,158.006
C04965=1034.050,135.664,399.865,169.388,42.536,158.006
C04966=1034.044,135.416,399.885,169.386,42.536,158.006
C04967=1034.038,135.167,399.907,169.383,42.537,158.006
C04968=1034.032,134.917,399.928,169.380,42.538,158.006
C04969=1034.026,134.669,399.948,169.378,42.539,158.006
C04970=1034.019,134.420,399.970,169.375,42.540,158.006
C04971=1034.013,134.171,399.990,169.373,42.540,158.006
C04972=1034.007,133.922,400.012,169.370,42.542,158.006
C04973=1034.001,133.672,400.033,169.368,42.543,158.006
C04974=1033.995,133.424,400.053,169.366,42.543,158.006
C04975=1033.989,133.174,400.075,169.363,42.544,158.006
C04976=1033.983,132.926,400.095,169.361,42.545,158.006
C04977=1033.977,132.676,400.116,169.358,42.546,158.006
C04978=1033.971,132.427,400.138,169.356,42.547,158.006
C04979=1033.965,132.178,400.158,169.353,42.548,158.006
C04980=1033.959,131.929,400.180,169.350,42.549,158.006
C04981=1033.953,131.680,400.200,169.349,42.550,158.006
C04982=1033.946,131.431,400.221,169.345,42.550,158.006
C04983=1033.941,131.182,400.242,169.344,42.551,158.006
C04984=1033.934,130.933,400.263,169.341,42.552,158.006
C04985=1033.928,130.683,400.284,169.339,42.553,158.006
C04986=1033.922,130.435,400.304,169.336,42.554,158.006
C04987=1033.916,130.185,400.325,169.333,42.555,158.006
C04988=1033.910,129.937,400.346,169.331,42.556,158.006
C04989=1033.903,129.688,400.366,169.328,42.557,158.006
C04990=1033.897,129.438,400.387,169.326,42.558,158.006
C04991=1033.891,129.190,400.408,169.324,42.559,158.006
C04992=1033.885,128.940,400.428,169.321,42.560,158.006
C04993=1033.878,128.692,400.449,169.319,42.561,158.006
C04994=1033.872,128.442,400.470,169.316,42.562,158.006
C04995=1033.866,128.193,400.490,169.313,42.563,158.006
C04996=1033.859,127.944,400.511,169.311,42.564,158.006
C04997=1033.854,127.695,400.532,169.308,42.565,158.006
C04998=1033.848,127.446,400.552,169.307,42.566,158.006
C04999=1033.841,127.197,400.573,169.304,42.567,158.006
C05000=1033.835,126.948,400.593,169.302,42.568,158.006
C05001=1033.829,126.698,400.614,169.299,42.569,158.006
C05002=1033.823,126.450,400.634,169.296,42.570,158.006
C05003=1033.816,126.200,400.655,169.294,42.571,158.006
C05004=1033.811,125.951,400.675,169.291,42.572,158.006
C05005=1033.804,125.702,400.696,169.290,42.573,158.006
C05006=1033.798,125.454,400.716,169.287,42.574,158.006
C05007=1033.791,125.204,400.737,169.284,42.575,158.006
C05008=1033.784,124.919,400.760,169.282,42.576,158.006
C05009=1033.777,124.633,400.784,169.279,42.577,158.007
C05010=1033.770,124.348,400.808,169.276,42.578,158.007
C05011=1033.763,124.063,400.831,169.273,42.579,158.007
C05012=1033.757,123.814,400.851,169.271,42.580,158.007
C05013=1033.751,123.564,400.872,169.269,42.581,158.007
C05014=1033.745,123.315,400.892,169.266,42.582,158.007
C05015=1033.739,123.067,400.913,169.264,42.583,158.007
C05016=1033.732,122.817,400.933,169.261,42.584,158.007
C05017=1033.726,122.569,400.953,169.258,42.585,158.007
C05018=1033.721,122.319,400.974,169.256,42.586,158.007
C05019=1033.715,122.070,400.994,169.254,42.587,158.007
C05020=1033.708,121.820,401.014,169.252,42.588,158.007
C05021=1033.702,121.572,401.035,169.249,42.589,158.007
C05022=1033.696,121.322,401.056,169.247,42.590,158.007
C05023=1033.690,121.074,401.076,169.244,42.591,158.007
C05024=1033.684,120.825,401.096,169.242,42.592,158.007
C05025=1033.677,120.575,401.116,169.239,42.593,158.007
C05026=1033.672,120.326,401.137,169.237,42.594,158.007
C05027=1033.665,120.077,401.157,169.235,42.595,158.007
C05028=1033.659,119.828,401.178,169.233,42.596,158.007
C05029=1033.653,119.580,401.198,169.230,42.596,158.007
C05030=1033.647,119.330,401.218,169.228,42.597,158.007
C05031=1033.641,119.081,401.238,169.225,42.598,158.007
C05032=1033.635,118.831,401.259,169.223,42.599,158.007
C05033=1033.629,118.583,401.279,169.220,42.600,158.007
C05034=1033.623,118.334,401.299,169.218,42.601,158.007
C05035=1033.617,118.084,401.320,169.216,42.602,158.007
C05036=1033.611,117.835,401.340,169.213,42.603,158.007
C05037=1033.605,117.586,401.360,169.211,42.604,158.007
C05038=1033.599,117.337,401.380,169.208,42.605,158.007
C05039=1033.593,117.088,401.400,169.206,42.606,158.007
C05040=1033.587,116.839,401.420,169.203,42.607,158.007
C05041=1033.580,116.589,401.441,169.201,42.607,158.007
C05042=1033.575,116.340,401.461,169.199,42.608,158.007
C05043=1033.569,116.092,401.481,169.197,42.610,158.007
C05044=1033.563,115.842,401.502,169.195,42.611,158.007
C05045=1033.557,115.593,401.521,169.192,42.612,158.007
C05046=1033.551,115.344,401.541,169.190,42.613,158.007
C05047=1033.545,115.095,401.562,169.187,42.613,158.007
C05048=1033.539,114.846,401.582,169.185,42.614,158.007
C05049=1033.533,114.597,401.602,169.182,42.615,158.007
C05050=1033.527,114.348,401.622,169.181,42.616,158.007
C05051=1033.521,114.098,401.643,169.178,42.617,158.007
C05052=1033.515,113.849,401.663,169.176,42.618,158.007
C05053=1033.509,113.601,401.683,169.173,42.619,158.007
C05054=1033.502,113.351,401.703,169.171,42.620,158.007
C05055=1033.496,113.102,401.723,169.168,42.621,158.007
C05056=1033.490,112.854,401.743,169.166,42.622,158.007
C05057=1033.484,112.603,401.763,169.163,42.623,158.007
C05058=1033.478,112.355,401.783,169.162,42.624,158.007
C05059=1033.472,112.106,401.803,169.159,42.625,158.007
C05060=1033.466,111.857,401.823,169.157,42.626,158.007
C05061=1033.459,111.607,401.843,169.154,42.627,158.007
C05062=1033.454,111.358,401.862,169.152,42.628,158.008
C05063=1033.448,111.109,401.882,169.149,42.629,158.007
C05064=1033.441,110.860,401.903,169.147,42.630,158.007
C05065=1033.435,110.611,401.923,169.145,42.631,158.007
C05066=1033.430,110.361,401.942,169.143,42.632,158.008
C05067=1033.424,110.113,401.962,169.140,42.633,158.008
C05068=1033.417,109.863,401.982,169.138,42.634,158.008
C05069=1033.410,109.614,402.001,169.135,42.635,158.008
C05070=1033.404,109.365,402.021,169.133,42.636,158.008
C05071=1033.398,109.116,402.041,169.130,42.637,158.008
C05072=1033.391,108.831,402.063,169.128,42.638,158.008
C05073=1033.384,108.545,402.086,169.125,42.640,158.008
C05074=1033.377,108.259,402.108,169.122,42.641,158.008
C05075=1033.369,107.973,402.131,169.120,42.642,158.008
C05076=1033.363,107.724,402.151,169.117,42.643,158.008
C05077=1033.357,107.476,402.171,169.116,42.644,158.008
C05078=1033.352,107.226,402.190,169.113,42.645,158.008
C05079=1033.344,106.977,402.210,169.111,42.646,158.008
C05080=1033.338,106.728,402.230,169.108,42.647,158.008
C05081=1033.333,106.479,402.249,169.106,42.648,158.008
C05082=1033.327,106.230,402.269,169.103,42.649,158.008
C05083=1033.320,105.980,402.288,169.102,42.650,158.008
C05084=1033.314,105.731,402.308,169.099,42.652,158.008
C05085=1033.308,105.482,402.327,169.097,42.652,158.008
C05086=1033.302,105.233,402.347,169.094,42.654,158.008
C05087=1033.296,104.984,402.367,169.092,42.655,158.008
C05088=1033.289,104.734,402.386,169.089,42.656,158.008
C05089=1033.283,104.486,402.406,169.088,42.657,158.008
C05090=1033.277,104.236,402.425,169.085,42.658,158.008
C05091=1033.271,103.987,402.445,169.083,42.659,158.009
C05092=1033.265,103.738,402.464,169.080,42.660,158.009
C05093=1033.259,103.489,402.484,169.078,42.661,158.009
C05094=1033.253,103.239,402.503,169.075,42.662,158.009
C05095=1033.247,102.990,402.523,169.074,42.663,158.009
C05096=1033.240,102.741,402.542,169.071,42.664,158.009
C05097=1033.234,102.493,402.562,169.069,42.665,158.009
C05098=1033.229,102.243,402.581,169.066,42.666,158.009
C05099=1033.223,101.994,402.601,169.064,42.667,158.009
C05100=1033.216,101.745,402.620,169.061,42.668,158.009
C05101=1033.210,101.496,402.640,169.059,42.669,158.009
C05102=1033.204,101.246,402.659,169.057,42.670,158.009
C05103=1033.198,100.997,402.679,169.055,42.671,158.009
C05104=1033.191,100.748,402.698,169.053,42.672,158.009
C05105=1033.186,100.499,402.717,169.050,42.673,158.009
C05106=1033.180,100.250,402.737,169.048,42.674,158.009
C05107=1033.174,100.001,402.756,169.045,42.675,158.009
C05108=1033.167,99.751,402.775,169.043,42.676,158.009
C05109=1033.161,99.502,402.795,169.041,42.677,158.009
C05110=1033.155,99.253,402.814,169.039,42.678,158.009
C05111=1033.149,99.003,402.833,169.036,42.680,158.009
C05112=1033.142,98.755,402.853,169.034,42.681,158.009
C05113=1033.137,98.505,402.872,169.031,42.682,158.009
C05114=1033.130,98.256,402.890,169.030,42.683,158.009
C05115=1033.124,98.006,402.910,169.027,42.684,158.009
C05116=1033.117,97.758,402.929,169.025,42.685,158.009
C05117=1033.111,97.509,402.948,169.022,42.686,158.009
C05118=1033.105,97.259,402.967,169.020,42.687,158.010
C05119=1033.099,97.010,402.986,169.017,42.688,158.010
C05120=1033.093,96.761,403.006,169.016,42.689,158.010
C05121=1033.086,96.512,403.025,169.013,42.690,158.010
C05122=1033.080,96.263,403.044,169.011,42.691,158.010
C05123=1033.074,96.014,403.062,169.008,42.693,158.010
C05124=1033.068,95.765,403.082,169.006,42.693,158.010
C05125=1033.061,95.515,403.101,169.003,42.695,158.010
C05126=1033.055,95.265,403.121,169.002,42.696,158.010
C05127=1033.049,95.016,403.139,168.999,42.697,158.010
C05128=1033.043,94.767,403.159,168.997,42.698,158.010
C05129=1033.037,94.518,403.177,168.995,42.699,158.010
C05130=1033.031,94.269,403.197,168.992,42.700,158.010
C05131=1033.024,94.020,403.216,168.990,42.701,158.010
C05132=1033.019,93.770,403.235,168.988,42.703,158.010
C05133=1033.012,93.521,403.254,168.986,42.704,158.010
C05134=1033.006,93.272,403.272,168.983,42.705,158.010
C05135=1033.000,93.023,403.292,168.981,42.706,158.010
C05136=1032.995,92.801,403.309,168.979,42.707,158.010
C05137=1032.989,92.579,403.325,168.976,42.708,158.010
C05138=1032.983,92.357,403.343,168.975,42.709,158.010
C05139=1032.978,92.135,403.359,168.973,42.710,158.010
C05140=1032.973,91.913,403.377,168.971,42.711,158.011
C05141=1032.967,91.691,403.393,168.969,42.711,158.010
C05142=1032.961,91.469,403.411,168.966,42.712,158.010
C05143=1032.956,91.247,403.427,168.964,42.713,158.011
C05144=1032.948,90.906,403.454,168.962,42.715,158.011
C05145=1032.939,90.567,403.479,168.959,42.716,158.011
C05146=1032.932,90.227,403.505,168.955,42.717,158.011
C05147=1032.923,89.887,403.530,168.952,42.719,158.011
C05148=1032.916,89.638,403.549,168.949,42.720,158.011
C05149=1032.911,89.388,403.568,168.948,42.721,158.011
C05150=1032.904,89.139,403.587,168.945,42.722,158.011
C05151=1032.898,88.890,403.606,168.943,42.723,158.011
C05152=1032.891,88.641,403.624,168.940,42.725,158.011
C05153=1032.885,88.392,403.643,168.938,42.726,158.011
C05154=1032.878,88.143,403.662,168.937,42.727,158.011
C05155=1032.873,87.893,403.681,168.934,42.728,158.011
C05156=1032.867,87.643,403.699,168.932,42.729,158.011
C05157=1032.860,87.394,403.717,168.929,42.730,158.011
C05158=1032.854,87.145,403.736,168.927,42.731,158.011
C05159=1032.847,86.896,403.755,168.925,42.733,158.012
C05160=1032.841,86.647,403.773,168.923,42.734,158.012
C05161=1032.835,86.398,403.793,168.920,42.735,158.012
C05162=1032.829,86.148,403.811,168.918,42.736,158.012
C05163=1032.822,85.899,403.830,168.915,42.737,158.012
C05164=1032.817,85.650,403.848,168.913,42.738,158.012
C05165=1032.810,85.401,403.866,168.910,42.740,158.012
C05166=1032.804,85.152,403.885,168.909,42.741,158.012
C05167=1032.798,84.903,403.904,168.906,42.742,158.012
C05168=1032.792,84.653,403.923,168.904,42.743,158.012
C05169=1032.785,84.404,403.941,168.901,42.744,158.012
C05170=1032.779,84.155,403.959,168.899,42.745,158.012
C05171=1032.773,83.905,403.978,168.897,42.747,158.012
C05172=1032.766,83.656,403.997,168.895,42.747,158.012
C05173=1032.760,83.407,404.015,168.893,42.748,158.012
C05174=1032.754,83.158,404.034,168.890,42.750,158.012
C05175=1032.748,82.908,404.052,168.888,42.751,158.012
C05176=1032.742,82.660,404.071,168.886,42.752,158.012
C05177=1032.736,82.411,404.089,168.884,42.753,158.012
C05178=1032.730,82.161,404.108,168.881,42.755,158.012
C05179=1032.723,81.912,404.126,168.879,42.755,158.013
C05180=1032.717,81.663,404.145,168.876,42.757,158.013
C05181=1032.711,81.413,404.163,168.874,42.758,158.013
C05182=1032.705,81.163,404.182,168.872,42.759,158.013
C05183=1032.699,80.914,404.200,168.870,42.760,158.013
C05184=1032.693,80.666,404.219,168.868,42.761,158.013
C05185=1032.687,80.417,404.237,168.865,42.762,158.013
C05186=1032.680,80.167,404.255,168.863,42.763,158.013
C05187=1032.674,79.918,404.274,168.861,42.765,158.013
C05188=1032.668,79.669,404.293,168.859,42.766,158.013
C05189=1032.662,79.419,404.311,168.856,42.767,158.013
C05190=1032.656,79.170,404.329,168.854,42.768,158.013
C05191=1032.650,78.921,404.348,168.851,42.769,158.013
C05192=1032.644,78.671,404.366,168.849,42.770,158.013
C05193=1032.637,78.422,404.385,168.848,42.771,158.013
C05194=1032.631,78.173,404.403,168.845,42.772,158.013
C05195=1032.625,77.923,404.421,168.843,42.773,158.013
C05196=1032.619,77.675,404.439,168.840,42.774,158.013
C05197=1032.613,77.425,404.457,168.838,42.775,158.013
C05198=1032.606,77.176,404.476,168.835,42.776,158.013
C05199=1032.600,76.926,404.494,168.834,42.778,158.013
C05200=1032.593,76.641,404.515,168.831,42.779,158.013
C05201=1032.587,76.355,404.536,168.828,42.780,158.013
C05202=1032.579,76.069,404.557,168.825,42.782,158.014
C05203=1032.571,75.784,404.578,168.823,42.783,158.014
C05204=1032.565,75.534,404.596,168.821,42.784,158.014
C05205=1032.559,75.286,404.614,168.819,42.785,158.014
C05206=1032.553,75.036,404.632,168.816,42.786,158.014
C05207=1032.547,74.787,404.650,168.814,42.788,158.014
C05208=1032.540,74.538,404.668,168.812,42.789,158.014
C05209=1032.534,74.289,404.686,168.810,42.790,158.014
C05210=1032.528,74.040,404.704,168.807,42.791,158.014
C05211=1032.522,73.790,404.723,168.805,42.792,158.014
C05212=1032.516,73.541,404.741,168.802,42.793,158.014
C05213=1032.509,73.291,404.758,168.801,42.795,158.014
C05214=1032.503,73.042,404.777,168.798,42.796,158.014
C05215=1032.497,72.793,404.794,168.796,42.797,158.014
C05216=1032.490,72.544,404.813,168.793,42.798,158.014
C05217=1032.484,72.294,404.831,168.791,42.799,158.014
C05218=1032.478,72.044,404.849,168.788,42.800,158.014
C05219=1032.472,71.796,404.867,168.786,42.801,158.014
C05220=1032.466,71.546,404.885,168.785,42.803,158.015
C05221=1032.459,71.297,404.903,168.782,42.804,158.015
C05222=1032.453,71.048,404.920,168.780,42.805,158.015
C05223=1032.447,70.799,404.938,168.777,42.806,158.015
C05224=1032.441,70.550,404.957,168.775,42.807,158.015
C05225=1032.435,70.300,404.975,168.773,42.808,158.015
C05226=1032.429,70.051,404.992,168.771,42.809,158.015
C05227=1032.422,69.802,405.011,168.768,42.811,158.015
C05228=1032.416,69.552,405.029,168.766,42.812,158.015
C05229=1032.410,69.303,405.046,168.763,42.813,158.015
C05230=1032.404,69.053,405.064,168.762,42.814,158.015
C05231=1032.397,68.805,405.082,168.759,42.815,158.015
C05232=1032.391,68.555,405.100,168.757,42.816,158.015
C05233=1032.386,68.306,405.118,168.755,42.818,158.015
C05234=1032.379,68.056,405.135,168.752,42.819,158.015
C05235=1032.372,67.807,405.154,168.751,42.820,158.015
C05236=1032.367,67.558,405.171,168.748,42.821,158.015
C05237=1032.360,67.309,405.188,168.746,42.822,158.016
C05238=1032.354,67.059,405.206,168.743,42.824,158.016
C05239=1032.347,66.810,405.225,168.741,42.825,158.016
C05240=1032.341,66.561,405.242,168.739,42.826,158.016
C05241=1032.335,66.312,405.260,168.737,42.827,158.016
C05242=1032.329,66.062,405.278,168.734,42.828,158.016
C05243=1032.323,65.813,405.295,168.732,42.830,158.016
C05244=1032.316,65.563,405.313,168.729,42.831,158.016
C05245=1032.310,65.314,405.330,168.728,42.832,158.016
C05246=1032.304,65.065,405.348,168.725,42.833,158.016
C05247=1032.298,64.816,405.366,168.723,42.834,158.016
C05248=1032.291,64.566,405.384,168.720,42.835,158.016
C05249=1032.285,64.317,405.401,168.718,42.837,158.016
C05250=1032.278,64.068,405.419,168.716,42.838,158.016
C05251=1032.273,63.819,405.436,168.714,42.839,158.016
C05252=1032.267,63.569,405.454,168.712,42.840,158.016
C05253=1032.260,63.320,405.471,168.709,42.842,158.017
C05254=1032.253,63.070,405.489,168.706,42.843,158.017
C05255=1032.248,62.821,405.506,168.705,42.844,158.017
C05256=1032.241,62.572,405.524,168.702,42.846,158.017
C05257=1032.234,62.322,405.541,168.700,42.847,158.017
C05258=1032.228,62.073,405.559,168.697,42.848,158.017
C05259=1032.221,61.824,405.576,168.696,42.850,158.017
C05260=1032.215,61.575,405.593,168.693,42.851,158.017
C05261=1032.209,61.325,405.611,168.691,42.852,158.017
C05262=1032.202,61.076,405.628,168.688,42.854,158.017
C05263=1032.196,60.827,405.645,168.687,42.855,158.017
C05264=1032.188,60.541,405.665,168.684,42.856,158.017
C05265=1032.181,60.255,405.685,168.681,42.857,158.017
C05266=1032.174,59.969,405.705,168.678,42.859,158.017
C05267=1032.167,59.683,405.725,168.676,42.860,158.018
C05268=1032.161,59.434,405.742,168.674,42.861,158.018
C05269=1032.154,59.185,405.760,168.671,42.863,158.018
C05270=1032.148,58.935,405.777,168.669,42.864,158.018
C05271=1032.141,58.686,405.794,168.666,42.865,158.018
C05272=1032.135,58.437,405.812,168.665,42.866,158.018
C05273=1032.129,58.188,405.829,168.662,42.868,158.018
C05274=1032.122,57.939,405.846,168.660,42.869,158.018
C05275=1032.116,57.688,405.863,168.657,42.870,158.018
C05276=1032.110,57.439,405.880,168.656,42.872,158.018
C05277=1032.103,57.190,405.898,168.653,42.873,158.018
C05278=1032.097,56.941,405.915,168.651,42.874,158.018
C05279=1032.091,56.692,405.933,168.648,42.875,158.018
C05280=1032.085,56.443,405.950,168.646,42.877,158.019
C05281=1032.078,56.193,405.966,168.644,42.878,158.019
C05282=1032.072,55.943,405.984,168.642,42.879,158.019
C05283=1032.066,55.694,406.001,168.639,42.880,158.019
C05284=1032.059,55.445,406.018,168.637,42.882,158.019
C05285=1032.053,55.196,406.036,168.634,42.883,158.019
C05286=1032.047,54.946,406.053,168.633,42.884,158.019
C05287=1032.040,54.697,406.070,168.630,42.885,158.019
C05288=1032.034,54.448,406.087,168.628,42.887,158.019
C05289=1032.028,54.199,406.104,168.625,42.888,158.019
C05290=1032.021,53.949,406.121,168.623,42.889,158.019
C05291=1032.015,53.700,406.138,168.621,42.890,158.019
C05292=1032.009,53.450,406.156,168.619,42.892,158.019
C05293=1032.003,53.201,406.173,168.616,42.893,158.019
C05294=1031.996,52.951,406.190,168.614,42.894,158.019
C05295=1031.990,52.703,406.207,168.611,42.895,158.019
C05296=1031.984,52.453,406.225,168.610,42.897,158.020
C05297=1031.978,52.203,406.241,168.607,42.898,158.020
C05298=1031.971,51.954,406.258,168.605,42.899,158.020
C05299=1031.966,51.705,406.276,168.602,42.900,158.020
C05300=1031.959,51.455,406.292,168.600,42.901,158.020
C05301=1031.953,51.206,406.309,168.598,42.903,158.020
C05302=1031.947,50.957,406.326,168.596,42.904,158.020
C05303=1031.941,50.707,406.343,168.593,42.905,158.020
C05304=1031.934,50.458,406.360,168.591,42.906,158.020
C05305=1031.928,50.209,406.378,168.588,42.907,158.020
C05306=1031.922,49.960,406.394,168.587,42.909,158.020
C05307=1031.916,49.710,406.412,168.584,42.910,158.020
C05308=1031.909,49.461,406.429,168.582,42.911,158.020
C05309=1031.903,49.212,406.445,168.579,42.912,158.020
C05310=1031.897,48.962,406.463,168.577,42.913,158.020
C05311=1031.891,48.713,406.479,168.575,42.915,158.020
C05312=1031.884,48.463,406.497,168.573,42.916,158.020
C05313=1031.878,48.215,406.514,168.570,42.917,158.020
C05314=1031.873,47.965,406.531,168.568,42.918,158.020
C05315=1031.866,47.715,406.548,168.565,42.919,158.020
C05316=1031.860,47.466,406.564,168.564,42.920,158.021
C05317=1031.853,47.217,406.581,168.561,42.922,158.021
C05318=1031.848,46.968,406.599,168.559,42.923,158.021
C05319=1031.842,46.718,406.615,168.556,42.924,158.021
C05320=1031.835,46.469,406.633,168.554,42.925,158.021
C05321=1031.829,46.220,406.649,168.552,42.926,158.021
C05322=1031.823,45.970,406.666,168.550,42.927,158.021
C05323=1031.817,45.720,406.683,168.547,42.928,158.021
C05324=1031.811,45.472,406.700,168.545,42.930,158.021
C05325=1031.804,45.222,406.717,168.543,42.931,158.021
C05326=1031.799,44.973,406.734,168.541,42.932,158.021
C05327=1031.793,44.723,406.751,168.539,42.933,158.021
C05328=1031.785,44.438,406.770,168.536,42.934,158.021
C05329=1031.778,44.151,406.789,168.533,42.936,158.021
C05330=1031.771,43.865,406.809,168.530,42.937,158.021
C05331=1031.764,43.579,406.828,168.528,42.938,158.021
C05332=1031.759,43.329,406.845,168.526,42.939,158.021
C05333=1031.752,43.080,406.862,168.523,42.941,158.021
C05334=1031.746,42.830,406.878,168.521,42.942,158.022
C05335=1031.740,42.582,406.895,168.518,42.943,158.022
C05336=1031.733,42.332,406.912,168.517,42.944,158.022
C05337=1031.727,42.082,406.928,168.514,42.945,158.022
C05338=1031.721,41.834,406.945,168.512,42.947,158.022
C05339=1031.714,41.584,406.962,168.509,42.948,158.022
C05340=1031.708,41.334,406.978,168.507,42.949,158.022
C05341=1031.702,41.085,406.995,168.505,42.950,158.022
C05342=1031.696,40.835,407.011,168.503,42.952,158.022
C05343=1031.690,40.586,407.028,168.500,42.953,158.022
C05344=1031.684,40.337,407.044,168.498,42.954,158.022
C05345=1031.677,40.087,407.061,168.495,42.955,158.022
C05346=1031.671,39.838,407.078,168.493,42.957,158.022
C05347=1031.665,39.589,407.094,168.491,42.958,158.022
C05348=1031.659,39.340,407.111,168.488,42.959,158.022
C05349=1031.652,39.090,407.127,168.486,42.960,158.022
C05350=1031.646,38.840,407.144,168.484,42.962,158.022
C05351=1031.640,38.591,407.160,168.482,42.963,158.022
C05352=1031.633,38.342,407.177,168.479,42.964,158.023
C05353=1031.627,38.093,407.193,168.477,42.965,158.023
C05354=1031.621,37.843,407.209,168.474,42.966,158.023
C05355=1031.615,37.594,407.225,168.473,42.968,158.023
C05356=1031.608,37.344,407.242,168.470,42.969,158.023
C05357=1031.602,37.095,407.259,168.468,42.970,158.023
C05358=1031.596,36.846,407.275,168.465,42.971,158.023
C05359=1031.590,36.596,407.292,168.463,42.973,158.023
C05360=1031.583,36.346,407.308,168.461,42.974,158.023
C05361=1031.577,36.097,407.324,168.459,42.976,158.023
C05362=1031.571,35.848,407.340,168.456,42.977,158.023
C05363=1031.565,35.599,407.356,168.453,42.978,158.023
C05364=1031.558,35.349,407.372,168.452,42.980,158.023
C05365=1031.552,35.100,407.389,168.449,42.981,158.023
C05366=1031.546,34.850,407.405,168.447,42.982,158.023
C05367=1031.539,34.602,407.422,168.444,42.984,158.024
C05368=1031.532,34.352,407.438,168.442,42.985,158.024
C05369=1031.526,34.102,407.454,168.440,42.986,158.024
C05370=1031.520,33.853,407.470,168.437,42.987,158.024
C05371=1031.514,33.604,407.487,168.435,42.989,158.024
C05372=1031.507,33.354,407.503,168.432,42.990,158.024
C05373=1031.501,33.105,407.519,168.430,42.991,158.024
C05374=1031.495,32.855,407.535,168.428,42.993,158.024
C05375=1031.488,32.606,407.551,168.426,42.994,158.024
C05376=1031.482,32.357,407.567,168.423,42.995,158.024
C05377=1031.476,32.107,407.584,168.421,42.997,158.024
C05378=1031.470,31.858,407.600,168.419,42.998,158.024
C05379=1031.463,31.609,407.616,168.416,42.999,158.024
C05380=1031.457,31.359,407.632,168.414,43.000,158.024
C05381=1031.451,31.110,407.648,168.411,43.002,158.024
C05382=1031.445,30.861,407.664,168.409,43.003,158.024
C05383=1031.438,30.611,407.680,168.407,43.004,158.024
C05384=1031.432,30.361,407.697,168.405,43.006,158.025
C05385=1031.426,30.112,407.713,168.402,43.007,158.025
C05386=1031.420,29.862,407.728,168.400,43.008,158.025
C05387=1031.414,29.613,407.744,168.397,43.009,158.025
C05388=1031.408,29.364,407.760,168.395,43.011,158.025
C05389=1031.401,29.115,407.776,168.393,43.012,158.025
C05390=1031.395,28.865,407.793,168.390,43.013,158.025
C05391=1031.389,28.615,407.809,168.388,43.014,158.025
C05392=1031.382,28.330,407.827,168.386,43.016,158.025
C05393=1031.375,28.043,407.846,168.383,43.017,158.025
C05394=1031.367,27.757,407.864,168.380,43.019,158.025
C05395=1031.360,27.470,407.882,168.377,43.020,158.025
C05396=1031.353,27.221,407.898,168.375,43.022,158.025
C05397=1031.347,26.972,407.914,168.373,43.023,158.025
C05398=1031.341,26.722,407.929,168.370,43.024,158.025
C05399=1031.335,26.473,407.946,168.368,43.026,158.026
C05400=1031.328,26.224,407.961,168.365,43.027,158.026
C05401=1031.322,25.975,407.977,168.363,43.028,158.026
C05402=1031.316,25.725,407.992,168.361,43.030,158.026
C05403=1031.309,25.475,408.009,168.358,43.031,158.026
C05404=1031.303,25.226,408.025,168.357,43.032,158.026
C05405=1031.297,24.976,408.041,168.354,43.034,158.026
C05406=1031.290,24.727,408.056,168.351,43.035,158.026
C05407=1031.285,24.477,408.072,168.349,43.036,158.026
C05408=1031.278,24.228,408.088,168.346,43.038,158.026
C05409=1031.272,23.979,408.104,168.345,43.039,158.026
C05410=1031.265,23.729,408.119,168.342,43.040,158.026
C05411=1031.259,23.480,408.135,168.339,43.041,158.026
C05412=1031.253,23.231,408.151,168.337,43.042,158.026
C05413=1031.246,22.981,408.166,168.335,43.044,158.027
C05414=1031.241,22.732,408.182,168.333,43.045,158.027
C05415=1031.234,22.483,408.198,168.330,43.046,158.027
C05416=1031.228,22.233,408.213,168.327,43.048,158.027
C05417=1031.221,21.983,408.229,168.325,43.049,158.027
C05418=1031.215,21.733,408.245,168.323,43.050,158.027
C05419=1031.209,21.484,408.261,168.321,43.052,158.027
C05420=1031.203,21.235,408.277,168.318,43.053,158.027
C05421=1031.196,20.985,408.292,168.315,43.054,158.027
C05422=1031.190,20.736,408.308,168.314,43.056,158.027
C05423=1031.184,20.487,408.324,168.311,43.057,158.027
C05424=1031.177,20.237,408.339,168.309,43.058,158.027
C05425=1031.171,19.988,408.355,168.306,43.059,158.027
C05426=1031.165,19.738,408.370,168.303,43.061,158.027
C05427=1031.159,19.489,408.386,168.302,43.062,158.027
C05428=1031.153,19.239,408.401,168.299,43.063,158.027
C05429=1031.146,18.990,408.417,168.297,43.065,158.028
C05430=1031.140,18.740,408.432,168.294,43.066,158.028
C05431=1031.134,18.491,408.448,168.292,43.068,158.028
C05432=1031.127,18.242,408.463,168.290,43.069,158.028
C05433=1031.121,17.992,408.479,168.287,43.070,158.028
C05434=1031.115,17.743,408.494,168.284,43.072,158.028
C05435=1031.108,17.493,408.510,168.282,43.073,158.028
C05436=1031.102,17.244,408.525,168.280,43.074,158.028
C05437=1031.096,16.994,408.541,168.278,43.076,158.028
C05438=1031.089,16.745,408.556,168.275,43.077,158.028
C05439=1031.083,16.496,408.572,168.272,43.078,158.028
C05440=1031.078,16.247,408.587,168.271,43.080,158.028
C05441=1031.071,15.997,408.602,168.268,43.081,158.028
C05442=1031.065,15.748,408.617,168.265,43.082,158.028
C05443=1031.059,15.498,408.633,168.263,43.084,158.028
C05444=1031.052,15.249,408.649,168.260,43.085,158.028
C05445=1031.046,14.999,408.663,168.259,43.086,158.028
C05446=1031.039,14.750,408.679,168.256,43.088,158.029
C05447=1031.034,14.500,408.695,168.253,43.089,158.029
C05448=1031.027,14.250,408.710,168.251,43.090,158.029
C05449=1031.020,14.001,408.725,168.249,43.092,158.029
C05450=1031.015,13.751,408.741,168.246,43.093,158.029
C05451=1031.008,13.502,408.756,168.244,43.095,158.029
C05452=1031.002,13.252,408.771,168.241,43.096,158.029
C05453=1030.995,13.003,408.786,168.239,43.098,158.029
C05454=1030.989,12.753,408.801,168.237,43.099,158.029
C05455=1030.983,12.504,408.816,168.234,43.101,158.029
C05456=1030.976,12.219,408.834,168.231,43.102,158.029
C05457=1030.967,11.934,408.851,168.229,43.104,158.029
C05458=1030.960,11.650,408.868,168.226,43.105,158.030
C05459=1030.954,11.365,408.885,168.223,43.107,158.030
C05460=1030.947,11.116,408.900,168.221,43.109,158.030
C05461=1030.941,10.866,408.915,168.218,43.110,158.030
C05462=1030.934,10.616,408.930,168.216,43.111,158.030
C05463=1030.928,10.367,408.945,168.213,43.113,158.030
